    PROC StoreSlot_P04(num slot, num subType, num toolSel, num lenMM,
                       robtarget arcStart, robtarget arcEnd, robtarget approach, robtarget retract, robtarget trans)
        IF slot = 1 THEN
            P04W01_SubType := subType;
            P04W01_ToolSel := toolSel;
            P04W01_LenMM := lenMM;
            P04W01_ArcStart := arcStart;
            P04W01_ArcEnd := arcEnd;
            P04W01_Approach := approach;
            P04W01_Retract := retract;
            P04W01_Trans := trans;
            P04W01_Used := TRUE;
        ELSEIF slot = 2 THEN
            P04W02_SubType := subType;
            P04W02_ToolSel := toolSel;
            P04W02_LenMM := lenMM;
            P04W02_ArcStart := arcStart;
            P04W02_ArcEnd := arcEnd;
            P04W02_Approach := approach;
            P04W02_Retract := retract;
            P04W02_Trans := trans;
            P04W02_Used := TRUE;
        ELSEIF slot = 3 THEN
            P04W03_SubType := subType;
            P04W03_ToolSel := toolSel;
            P04W03_LenMM := lenMM;
            P04W03_ArcStart := arcStart;
            P04W03_ArcEnd := arcEnd;
            P04W03_Approach := approach;
            P04W03_Retract := retract;
            P04W03_Trans := trans;
            P04W03_Used := TRUE;
        ELSEIF slot = 4 THEN
            P04W04_SubType := subType;
            P04W04_ToolSel := toolSel;
            P04W04_LenMM := lenMM;
            P04W04_ArcStart := arcStart;
            P04W04_ArcEnd := arcEnd;
            P04W04_Approach := approach;
            P04W04_Retract := retract;
            P04W04_Trans := trans;
            P04W04_Used := TRUE;
        ELSEIF slot = 5 THEN
            P04W05_SubType := subType;
            P04W05_ToolSel := toolSel;
            P04W05_LenMM := lenMM;
            P04W05_ArcStart := arcStart;
            P04W05_ArcEnd := arcEnd;
            P04W05_Approach := approach;
            P04W05_Retract := retract;
            P04W05_Trans := trans;
            P04W05_Used := TRUE;
        ELSEIF slot = 6 THEN
            P04W06_SubType := subType;
            P04W06_ToolSel := toolSel;
            P04W06_LenMM := lenMM;
            P04W06_ArcStart := arcStart;
            P04W06_ArcEnd := arcEnd;
            P04W06_Approach := approach;
            P04W06_Retract := retract;
            P04W06_Trans := trans;
            P04W06_Used := TRUE;
        ELSEIF slot = 7 THEN
            P04W07_SubType := subType;
            P04W07_ToolSel := toolSel;
            P04W07_LenMM := lenMM;
            P04W07_ArcStart := arcStart;
            P04W07_ArcEnd := arcEnd;
            P04W07_Approach := approach;
            P04W07_Retract := retract;
            P04W07_Trans := trans;
            P04W07_Used := TRUE;
        ELSEIF slot = 8 THEN
            P04W08_SubType := subType;
            P04W08_ToolSel := toolSel;
            P04W08_LenMM := lenMM;
            P04W08_ArcStart := arcStart;
            P04W08_ArcEnd := arcEnd;
            P04W08_Approach := approach;
            P04W08_Retract := retract;
            P04W08_Trans := trans;
            P04W08_Used := TRUE;
        ELSEIF slot = 9 THEN
            P04W09_SubType := subType;
            P04W09_ToolSel := toolSel;
            P04W09_LenMM := lenMM;
            P04W09_ArcStart := arcStart;
            P04W09_ArcEnd := arcEnd;
            P04W09_Approach := approach;
            P04W09_Retract := retract;
            P04W09_Trans := trans;
            P04W09_Used := TRUE;
        ELSEIF slot = 10 THEN
            P04W10_SubType := subType;
            P04W10_ToolSel := toolSel;
            P04W10_LenMM := lenMM;
            P04W10_ArcStart := arcStart;
            P04W10_ArcEnd := arcEnd;
            P04W10_Approach := approach;
            P04W10_Retract := retract;
            P04W10_Trans := trans;
            P04W10_Used := TRUE;
        ELSEIF slot = 11 THEN
            P04W11_SubType := subType;
            P04W11_ToolSel := toolSel;
            P04W11_LenMM := lenMM;
            P04W11_ArcStart := arcStart;
            P04W11_ArcEnd := arcEnd;
            P04W11_Approach := approach;
            P04W11_Retract := retract;
            P04W11_Trans := trans;
            P04W11_Used := TRUE;
        ELSEIF slot = 12 THEN
            P04W12_SubType := subType;
            P04W12_ToolSel := toolSel;
            P04W12_LenMM := lenMM;
            P04W12_ArcStart := arcStart;
            P04W12_ArcEnd := arcEnd;
            P04W12_Approach := approach;
            P04W12_Retract := retract;
            P04W12_Trans := trans;
            P04W12_Used := TRUE;
        ELSEIF slot = 13 THEN
            P04W13_SubType := subType;
            P04W13_ToolSel := toolSel;
            P04W13_LenMM := lenMM;
            P04W13_ArcStart := arcStart;
            P04W13_ArcEnd := arcEnd;
            P04W13_Approach := approach;
            P04W13_Retract := retract;
            P04W13_Trans := trans;
            P04W13_Used := TRUE;
        ELSEIF slot = 14 THEN
            P04W14_SubType := subType;
            P04W14_ToolSel := toolSel;
            P04W14_LenMM := lenMM;
            P04W14_ArcStart := arcStart;
            P04W14_ArcEnd := arcEnd;
            P04W14_Approach := approach;
            P04W14_Retract := retract;
            P04W14_Trans := trans;
            P04W14_Used := TRUE;
        ELSEIF slot = 15 THEN
            P04W15_SubType := subType;
            P04W15_ToolSel := toolSel;
            P04W15_LenMM := lenMM;
            P04W15_ArcStart := arcStart;
            P04W15_ArcEnd := arcEnd;
            P04W15_Approach := approach;
            P04W15_Retract := retract;
            P04W15_Trans := trans;
            P04W15_Used := TRUE;
        ELSEIF slot = 16 THEN
            P04W16_SubType := subType;
            P04W16_ToolSel := toolSel;
            P04W16_LenMM := lenMM;
            P04W16_ArcStart := arcStart;
            P04W16_ArcEnd := arcEnd;
            P04W16_Approach := approach;
            P04W16_Retract := retract;
            P04W16_Trans := trans;
            P04W16_Used := TRUE;
        ELSEIF slot = 17 THEN
            P04W17_SubType := subType;
            P04W17_ToolSel := toolSel;
            P04W17_LenMM := lenMM;
            P04W17_ArcStart := arcStart;
            P04W17_ArcEnd := arcEnd;
            P04W17_Approach := approach;
            P04W17_Retract := retract;
            P04W17_Trans := trans;
            P04W17_Used := TRUE;
        ELSEIF slot = 18 THEN
            P04W18_SubType := subType;
            P04W18_ToolSel := toolSel;
            P04W18_LenMM := lenMM;
            P04W18_ArcStart := arcStart;
            P04W18_ArcEnd := arcEnd;
            P04W18_Approach := approach;
            P04W18_Retract := retract;
            P04W18_Trans := trans;
            P04W18_Used := TRUE;
        ELSEIF slot = 19 THEN
            P04W19_SubType := subType;
            P04W19_ToolSel := toolSel;
            P04W19_LenMM := lenMM;
            P04W19_ArcStart := arcStart;
            P04W19_ArcEnd := arcEnd;
            P04W19_Approach := approach;
            P04W19_Retract := retract;
            P04W19_Trans := trans;
            P04W19_Used := TRUE;
        ELSEIF slot = 20 THEN
            P04W20_SubType := subType;
            P04W20_ToolSel := toolSel;
            P04W20_LenMM := lenMM;
            P04W20_ArcStart := arcStart;
            P04W20_ArcEnd := arcEnd;
            P04W20_Approach := approach;
            P04W20_Retract := retract;
            P04W20_Trans := trans;
            P04W20_Used := TRUE;
        ELSEIF slot = 21 THEN
            P04W21_SubType := subType;
            P04W21_ToolSel := toolSel;
            P04W21_LenMM := lenMM;
            P04W21_ArcStart := arcStart;
            P04W21_ArcEnd := arcEnd;
            P04W21_Approach := approach;
            P04W21_Retract := retract;
            P04W21_Trans := trans;
            P04W21_Used := TRUE;
        ELSEIF slot = 22 THEN
            P04W22_SubType := subType;
            P04W22_ToolSel := toolSel;
            P04W22_LenMM := lenMM;
            P04W22_ArcStart := arcStart;
            P04W22_ArcEnd := arcEnd;
            P04W22_Approach := approach;
            P04W22_Retract := retract;
            P04W22_Trans := trans;
            P04W22_Used := TRUE;
        ELSEIF slot = 23 THEN
            P04W23_SubType := subType;
            P04W23_ToolSel := toolSel;
            P04W23_LenMM := lenMM;
            P04W23_ArcStart := arcStart;
            P04W23_ArcEnd := arcEnd;
            P04W23_Approach := approach;
            P04W23_Retract := retract;
            P04W23_Trans := trans;
            P04W23_Used := TRUE;
        ELSEIF slot = 24 THEN
            P04W24_SubType := subType;
            P04W24_ToolSel := toolSel;
            P04W24_LenMM := lenMM;
            P04W24_ArcStart := arcStart;
            P04W24_ArcEnd := arcEnd;
            P04W24_Approach := approach;
            P04W24_Retract := retract;
            P04W24_Trans := trans;
            P04W24_Used := TRUE;
        ELSEIF slot = 25 THEN
            P04W25_SubType := subType;
            P04W25_ToolSel := toolSel;
            P04W25_LenMM := lenMM;
            P04W25_ArcStart := arcStart;
            P04W25_ArcEnd := arcEnd;
            P04W25_Approach := approach;
            P04W25_Retract := retract;
            P04W25_Trans := trans;
            P04W25_Used := TRUE;
        ELSEIF slot = 26 THEN
            P04W26_SubType := subType;
            P04W26_ToolSel := toolSel;
            P04W26_LenMM := lenMM;
            P04W26_ArcStart := arcStart;
            P04W26_ArcEnd := arcEnd;
            P04W26_Approach := approach;
            P04W26_Retract := retract;
            P04W26_Trans := trans;
            P04W26_Used := TRUE;
        ELSEIF slot = 27 THEN
            P04W27_SubType := subType;
            P04W27_ToolSel := toolSel;
            P04W27_LenMM := lenMM;
            P04W27_ArcStart := arcStart;
            P04W27_ArcEnd := arcEnd;
            P04W27_Approach := approach;
            P04W27_Retract := retract;
            P04W27_Trans := trans;
            P04W27_Used := TRUE;
        ELSEIF slot = 28 THEN
            P04W28_SubType := subType;
            P04W28_ToolSel := toolSel;
            P04W28_LenMM := lenMM;
            P04W28_ArcStart := arcStart;
            P04W28_ArcEnd := arcEnd;
            P04W28_Approach := approach;
            P04W28_Retract := retract;
            P04W28_Trans := trans;
            P04W28_Used := TRUE;
        ELSEIF slot = 29 THEN
            P04W29_SubType := subType;
            P04W29_ToolSel := toolSel;
            P04W29_LenMM := lenMM;
            P04W29_ArcStart := arcStart;
            P04W29_ArcEnd := arcEnd;
            P04W29_Approach := approach;
            P04W29_Retract := retract;
            P04W29_Trans := trans;
            P04W29_Used := TRUE;
        ELSEIF slot = 30 THEN
            P04W30_SubType := subType;
            P04W30_ToolSel := toolSel;
            P04W30_LenMM := lenMM;
            P04W30_ArcStart := arcStart;
            P04W30_ArcEnd := arcEnd;
            P04W30_Approach := approach;
            P04W30_Retract := retract;
            P04W30_Trans := trans;
            P04W30_Used := TRUE;
        ELSE
            TPWrite "Invalid weld slot.";
        ENDIF
    ENDPROC

    PROC LoadSlot_P04(num slot, VAR bool used, VAR num subType, VAR num toolSel, VAR num lenMM,
                       VAR robtarget arcStart, VAR robtarget arcEnd, VAR robtarget approach, VAR robtarget retract, VAR robtarget trans)
        IF slot = 1 THEN
            used := P04W01_Used;
            subType := P04W01_SubType;
            toolSel := P04W01_ToolSel;
            lenMM := P04W01_LenMM;
            arcStart := P04W01_ArcStart;
            arcEnd := P04W01_ArcEnd;
            approach := P04W01_Approach;
            retract := P04W01_Retract;
            trans := P04W01_Trans;
        ELSEIF slot = 2 THEN
            used := P04W02_Used;
            subType := P04W02_SubType;
            toolSel := P04W02_ToolSel;
            lenMM := P04W02_LenMM;
            arcStart := P04W02_ArcStart;
            arcEnd := P04W02_ArcEnd;
            approach := P04W02_Approach;
            retract := P04W02_Retract;
            trans := P04W02_Trans;
        ELSEIF slot = 3 THEN
            used := P04W03_Used;
            subType := P04W03_SubType;
            toolSel := P04W03_ToolSel;
            lenMM := P04W03_LenMM;
            arcStart := P04W03_ArcStart;
            arcEnd := P04W03_ArcEnd;
            approach := P04W03_Approach;
            retract := P04W03_Retract;
            trans := P04W03_Trans;
        ELSEIF slot = 4 THEN
            used := P04W04_Used;
            subType := P04W04_SubType;
            toolSel := P04W04_ToolSel;
            lenMM := P04W04_LenMM;
            arcStart := P04W04_ArcStart;
            arcEnd := P04W04_ArcEnd;
            approach := P04W04_Approach;
            retract := P04W04_Retract;
            trans := P04W04_Trans;
        ELSEIF slot = 5 THEN
            used := P04W05_Used;
            subType := P04W05_SubType;
            toolSel := P04W05_ToolSel;
            lenMM := P04W05_LenMM;
            arcStart := P04W05_ArcStart;
            arcEnd := P04W05_ArcEnd;
            approach := P04W05_Approach;
            retract := P04W05_Retract;
            trans := P04W05_Trans;
        ELSEIF slot = 6 THEN
            used := P04W06_Used;
            subType := P04W06_SubType;
            toolSel := P04W06_ToolSel;
            lenMM := P04W06_LenMM;
            arcStart := P04W06_ArcStart;
            arcEnd := P04W06_ArcEnd;
            approach := P04W06_Approach;
            retract := P04W06_Retract;
            trans := P04W06_Trans;
        ELSEIF slot = 7 THEN
            used := P04W07_Used;
            subType := P04W07_SubType;
            toolSel := P04W07_ToolSel;
            lenMM := P04W07_LenMM;
            arcStart := P04W07_ArcStart;
            arcEnd := P04W07_ArcEnd;
            approach := P04W07_Approach;
            retract := P04W07_Retract;
            trans := P04W07_Trans;
        ELSEIF slot = 8 THEN
            used := P04W08_Used;
            subType := P04W08_SubType;
            toolSel := P04W08_ToolSel;
            lenMM := P04W08_LenMM;
            arcStart := P04W08_ArcStart;
            arcEnd := P04W08_ArcEnd;
            approach := P04W08_Approach;
            retract := P04W08_Retract;
            trans := P04W08_Trans;
        ELSEIF slot = 9 THEN
            used := P04W09_Used;
            subType := P04W09_SubType;
            toolSel := P04W09_ToolSel;
            lenMM := P04W09_LenMM;
            arcStart := P04W09_ArcStart;
            arcEnd := P04W09_ArcEnd;
            approach := P04W09_Approach;
            retract := P04W09_Retract;
            trans := P04W09_Trans;
        ELSEIF slot = 10 THEN
            used := P04W10_Used;
            subType := P04W10_SubType;
            toolSel := P04W10_ToolSel;
            lenMM := P04W10_LenMM;
            arcStart := P04W10_ArcStart;
            arcEnd := P04W10_ArcEnd;
            approach := P04W10_Approach;
            retract := P04W10_Retract;
            trans := P04W10_Trans;
        ELSEIF slot = 11 THEN
            used := P04W11_Used;
            subType := P04W11_SubType;
            toolSel := P04W11_ToolSel;
            lenMM := P04W11_LenMM;
            arcStart := P04W11_ArcStart;
            arcEnd := P04W11_ArcEnd;
            approach := P04W11_Approach;
            retract := P04W11_Retract;
            trans := P04W11_Trans;
        ELSEIF slot = 12 THEN
            used := P04W12_Used;
            subType := P04W12_SubType;
            toolSel := P04W12_ToolSel;
            lenMM := P04W12_LenMM;
            arcStart := P04W12_ArcStart;
            arcEnd := P04W12_ArcEnd;
            approach := P04W12_Approach;
            retract := P04W12_Retract;
            trans := P04W12_Trans;
        ELSEIF slot = 13 THEN
            used := P04W13_Used;
            subType := P04W13_SubType;
            toolSel := P04W13_ToolSel;
            lenMM := P04W13_LenMM;
            arcStart := P04W13_ArcStart;
            arcEnd := P04W13_ArcEnd;
            approach := P04W13_Approach;
            retract := P04W13_Retract;
            trans := P04W13_Trans;
        ELSEIF slot = 14 THEN
            used := P04W14_Used;
            subType := P04W14_SubType;
            toolSel := P04W14_ToolSel;
            lenMM := P04W14_LenMM;
            arcStart := P04W14_ArcStart;
            arcEnd := P04W14_ArcEnd;
            approach := P04W14_Approach;
            retract := P04W14_Retract;
            trans := P04W14_Trans;
        ELSEIF slot = 15 THEN
            used := P04W15_Used;
            subType := P04W15_SubType;
            toolSel := P04W15_ToolSel;
            lenMM := P04W15_LenMM;
            arcStart := P04W15_ArcStart;
            arcEnd := P04W15_ArcEnd;
            approach := P04W15_Approach;
            retract := P04W15_Retract;
            trans := P04W15_Trans;
        ELSEIF slot = 16 THEN
            used := P04W16_Used;
            subType := P04W16_SubType;
            toolSel := P04W16_ToolSel;
            lenMM := P04W16_LenMM;
            arcStart := P04W16_ArcStart;
            arcEnd := P04W16_ArcEnd;
            approach := P04W16_Approach;
            retract := P04W16_Retract;
            trans := P04W16_Trans;
        ELSEIF slot = 17 THEN
            used := P04W17_Used;
            subType := P04W17_SubType;
            toolSel := P04W17_ToolSel;
            lenMM := P04W17_LenMM;
            arcStart := P04W17_ArcStart;
            arcEnd := P04W17_ArcEnd;
            approach := P04W17_Approach;
            retract := P04W17_Retract;
            trans := P04W17_Trans;
        ELSEIF slot = 18 THEN
            used := P04W18_Used;
            subType := P04W18_SubType;
            toolSel := P04W18_ToolSel;
            lenMM := P04W18_LenMM;
            arcStart := P04W18_ArcStart;
            arcEnd := P04W18_ArcEnd;
            approach := P04W18_Approach;
            retract := P04W18_Retract;
            trans := P04W18_Trans;
        ELSEIF slot = 19 THEN
            used := P04W19_Used;
            subType := P04W19_SubType;
            toolSel := P04W19_ToolSel;
            lenMM := P04W19_LenMM;
            arcStart := P04W19_ArcStart;
            arcEnd := P04W19_ArcEnd;
            approach := P04W19_Approach;
            retract := P04W19_Retract;
            trans := P04W19_Trans;
        ELSEIF slot = 20 THEN
            used := P04W20_Used;
            subType := P04W20_SubType;
            toolSel := P04W20_ToolSel;
            lenMM := P04W20_LenMM;
            arcStart := P04W20_ArcStart;
            arcEnd := P04W20_ArcEnd;
            approach := P04W20_Approach;
            retract := P04W20_Retract;
            trans := P04W20_Trans;
        ELSEIF slot = 21 THEN
            used := P04W21_Used;
            subType := P04W21_SubType;
            toolSel := P04W21_ToolSel;
            lenMM := P04W21_LenMM;
            arcStart := P04W21_ArcStart;
            arcEnd := P04W21_ArcEnd;
            approach := P04W21_Approach;
            retract := P04W21_Retract;
            trans := P04W21_Trans;
        ELSEIF slot = 22 THEN
            used := P04W22_Used;
            subType := P04W22_SubType;
            toolSel := P04W22_ToolSel;
            lenMM := P04W22_LenMM;
            arcStart := P04W22_ArcStart;
            arcEnd := P04W22_ArcEnd;
            approach := P04W22_Approach;
            retract := P04W22_Retract;
            trans := P04W22_Trans;
        ELSEIF slot = 23 THEN
            used := P04W23_Used;
            subType := P04W23_SubType;
            toolSel := P04W23_ToolSel;
            lenMM := P04W23_LenMM;
            arcStart := P04W23_ArcStart;
            arcEnd := P04W23_ArcEnd;
            approach := P04W23_Approach;
            retract := P04W23_Retract;
            trans := P04W23_Trans;
        ELSEIF slot = 24 THEN
            used := P04W24_Used;
            subType := P04W24_SubType;
            toolSel := P04W24_ToolSel;
            lenMM := P04W24_LenMM;
            arcStart := P04W24_ArcStart;
            arcEnd := P04W24_ArcEnd;
            approach := P04W24_Approach;
            retract := P04W24_Retract;
            trans := P04W24_Trans;
        ELSEIF slot = 25 THEN
            used := P04W25_Used;
            subType := P04W25_SubType;
            toolSel := P04W25_ToolSel;
            lenMM := P04W25_LenMM;
            arcStart := P04W25_ArcStart;
            arcEnd := P04W25_ArcEnd;
            approach := P04W25_Approach;
            retract := P04W25_Retract;
            trans := P04W25_Trans;
        ELSEIF slot = 26 THEN
            used := P04W26_Used;
            subType := P04W26_SubType;
            toolSel := P04W26_ToolSel;
            lenMM := P04W26_LenMM;
            arcStart := P04W26_ArcStart;
            arcEnd := P04W26_ArcEnd;
            approach := P04W26_Approach;
            retract := P04W26_Retract;
            trans := P04W26_Trans;
        ELSEIF slot = 27 THEN
            used := P04W27_Used;
            subType := P04W27_SubType;
            toolSel := P04W27_ToolSel;
            lenMM := P04W27_LenMM;
            arcStart := P04W27_ArcStart;
            arcEnd := P04W27_ArcEnd;
            approach := P04W27_Approach;
            retract := P04W27_Retract;
            trans := P04W27_Trans;
        ELSEIF slot = 28 THEN
            used := P04W28_Used;
            subType := P04W28_SubType;
            toolSel := P04W28_ToolSel;
            lenMM := P04W28_LenMM;
            arcStart := P04W28_ArcStart;
            arcEnd := P04W28_ArcEnd;
            approach := P04W28_Approach;
            retract := P04W28_Retract;
            trans := P04W28_Trans;
        ELSEIF slot = 29 THEN
            used := P04W29_Used;
            subType := P04W29_SubType;
            toolSel := P04W29_ToolSel;
            lenMM := P04W29_LenMM;
            arcStart := P04W29_ArcStart;
            arcEnd := P04W29_ArcEnd;
            approach := P04W29_Approach;
            retract := P04W29_Retract;
            trans := P04W29_Trans;
        ELSEIF slot = 30 THEN
            used := P04W30_Used;
            subType := P04W30_SubType;
            toolSel := P04W30_ToolSel;
            lenMM := P04W30_LenMM;
            arcStart := P04W30_ArcStart;
            arcEnd := P04W30_ArcEnd;
            approach := P04W30_Approach;
            retract := P04W30_Retract;
            trans := P04W30_Trans;
        ELSE
            used := FALSE;
        ENDIF
    ENDPROC

    PROC ClearSlot_P04(num slot)
        IF slot = 1 THEN
            P04W01_Used := FALSE;
            P04W01_SubType := 0;
            P04W01_ToolSel := 0;
            P04W01_LenMM := 0;
            P04W01_ArcStart := [[0,0,0],[1,0,0,0],[0,0,0,0],[9E9,9E9,9E9,9E9,9E9,9E9]];
            P04W01_ArcEnd := [[0,0,0],[1,0,0,0],[0,0,0,0],[9E9,9E9,9E9,9E9,9E9,9E9]];
            P04W01_Approach := [[0,0,0],[1,0,0,0],[0,0,0,0],[9E9,9E9,9E9,9E9,9E9,9E9]];
            P04W01_Retract := [[0,0,0],[1,0,0,0],[0,0,0,0],[9E9,9E9,9E9,9E9,9E9,9E9]];
            P04W01_Trans := [[0,0,0],[1,0,0,0],[0,0,0,0],[9E9,9E9,9E9,9E9,9E9,9E9]];
        ELSEIF slot = 2 THEN
            P04W02_Used := FALSE;
            P04W02_SubType := 0;
            P04W02_ToolSel := 0;
            P04W02_LenMM := 0;
            P04W02_ArcStart := [[0,0,0],[1,0,0,0],[0,0,0,0],[9E9,9E9,9E9,9E9,9E9,9E9]];
            P04W02_ArcEnd := [[0,0,0],[1,0,0,0],[0,0,0,0],[9E9,9E9,9E9,9E9,9E9,9E9]];
            P04W02_Approach := [[0,0,0],[1,0,0,0],[0,0,0,0],[9E9,9E9,9E9,9E9,9E9,9E9]];
            P04W02_Retract := [[0,0,0],[1,0,0,0],[0,0,0,0],[9E9,9E9,9E9,9E9,9E9,9E9]];
            P04W02_Trans := [[0,0,0],[1,0,0,0],[0,0,0,0],[9E9,9E9,9E9,9E9,9E9,9E9]];
        ELSEIF slot = 3 THEN
            P04W03_Used := FALSE;
            P04W03_SubType := 0;
            P04W03_ToolSel := 0;
            P04W03_LenMM := 0;
            P04W03_ArcStart := [[0,0,0],[1,0,0,0],[0,0,0,0],[9E9,9E9,9E9,9E9,9E9,9E9]];
            P04W03_ArcEnd := [[0,0,0],[1,0,0,0],[0,0,0,0],[9E9,9E9,9E9,9E9,9E9,9E9]];
            P04W03_Approach := [[0,0,0],[1,0,0,0],[0,0,0,0],[9E9,9E9,9E9,9E9,9E9,9E9]];
            P04W03_Retract := [[0,0,0],[1,0,0,0],[0,0,0,0],[9E9,9E9,9E9,9E9,9E9,9E9]];
            P04W03_Trans := [[0,0,0],[1,0,0,0],[0,0,0,0],[9E9,9E9,9E9,9E9,9E9,9E9]];
        ELSEIF slot = 4 THEN
            P04W04_Used := FALSE;
            P04W04_SubType := 0;
            P04W04_ToolSel := 0;
            P04W04_LenMM := 0;
            P04W04_ArcStart := [[0,0,0],[1,0,0,0],[0,0,0,0],[9E9,9E9,9E9,9E9,9E9,9E9]];
            P04W04_ArcEnd := [[0,0,0],[1,0,0,0],[0,0,0,0],[9E9,9E9,9E9,9E9,9E9,9E9]];
            P04W04_Approach := [[0,0,0],[1,0,0,0],[0,0,0,0],[9E9,9E9,9E9,9E9,9E9,9E9]];
            P04W04_Retract := [[0,0,0],[1,0,0,0],[0,0,0,0],[9E9,9E9,9E9,9E9,9E9,9E9]];
            P04W04_Trans := [[0,0,0],[1,0,0,0],[0,0,0,0],[9E9,9E9,9E9,9E9,9E9,9E9]];
        ELSEIF slot = 5 THEN
            P04W05_Used := FALSE;
            P04W05_SubType := 0;
            P04W05_ToolSel := 0;
            P04W05_LenMM := 0;
            P04W05_ArcStart := [[0,0,0],[1,0,0,0],[0,0,0,0],[9E9,9E9,9E9,9E9,9E9,9E9]];
            P04W05_ArcEnd := [[0,0,0],[1,0,0,0],[0,0,0,0],[9E9,9E9,9E9,9E9,9E9,9E9]];
            P04W05_Approach := [[0,0,0],[1,0,0,0],[0,0,0,0],[9E9,9E9,9E9,9E9,9E9,9E9]];
            P04W05_Retract := [[0,0,0],[1,0,0,0],[0,0,0,0],[9E9,9E9,9E9,9E9,9E9,9E9]];
            P04W05_Trans := [[0,0,0],[1,0,0,0],[0,0,0,0],[9E9,9E9,9E9,9E9,9E9,9E9]];
        ELSEIF slot = 6 THEN
            P04W06_Used := FALSE;
            P04W06_SubType := 0;
            P04W06_ToolSel := 0;
            P04W06_LenMM := 0;
            P04W06_ArcStart := [[0,0,0],[1,0,0,0],[0,0,0,0],[9E9,9E9,9E9,9E9,9E9,9E9]];
            P04W06_ArcEnd := [[0,0,0],[1,0,0,0],[0,0,0,0],[9E9,9E9,9E9,9E9,9E9,9E9]];
            P04W06_Approach := [[0,0,0],[1,0,0,0],[0,0,0,0],[9E9,9E9,9E9,9E9,9E9,9E9]];
            P04W06_Retract := [[0,0,0],[1,0,0,0],[0,0,0,0],[9E9,9E9,9E9,9E9,9E9,9E9]];
            P04W06_Trans := [[0,0,0],[1,0,0,0],[0,0,0,0],[9E9,9E9,9E9,9E9,9E9,9E9]];
        ELSEIF slot = 7 THEN
            P04W07_Used := FALSE;
            P04W07_SubType := 0;
            P04W07_ToolSel := 0;
            P04W07_LenMM := 0;
            P04W07_ArcStart := [[0,0,0],[1,0,0,0],[0,0,0,0],[9E9,9E9,9E9,9E9,9E9,9E9]];
            P04W07_ArcEnd := [[0,0,0],[1,0,0,0],[0,0,0,0],[9E9,9E9,9E9,9E9,9E9,9E9]];
            P04W07_Approach := [[0,0,0],[1,0,0,0],[0,0,0,0],[9E9,9E9,9E9,9E9,9E9,9E9]];
            P04W07_Retract := [[0,0,0],[1,0,0,0],[0,0,0,0],[9E9,9E9,9E9,9E9,9E9,9E9]];
            P04W07_Trans := [[0,0,0],[1,0,0,0],[0,0,0,0],[9E9,9E9,9E9,9E9,9E9,9E9]];
        ELSEIF slot = 8 THEN
            P04W08_Used := FALSE;
            P04W08_SubType := 0;
            P04W08_ToolSel := 0;
            P04W08_LenMM := 0;
            P04W08_ArcStart := [[0,0,0],[1,0,0,0],[0,0,0,0],[9E9,9E9,9E9,9E9,9E9,9E9]];
            P04W08_ArcEnd := [[0,0,0],[1,0,0,0],[0,0,0,0],[9E9,9E9,9E9,9E9,9E9,9E9]];
            P04W08_Approach := [[0,0,0],[1,0,0,0],[0,0,0,0],[9E9,9E9,9E9,9E9,9E9,9E9]];
            P04W08_Retract := [[0,0,0],[1,0,0,0],[0,0,0,0],[9E9,9E9,9E9,9E9,9E9,9E9]];
            P04W08_Trans := [[0,0,0],[1,0,0,0],[0,0,0,0],[9E9,9E9,9E9,9E9,9E9,9E9]];
        ELSEIF slot = 9 THEN
            P04W09_Used := FALSE;
            P04W09_SubType := 0;
            P04W09_ToolSel := 0;
            P04W09_LenMM := 0;
            P04W09_ArcStart := [[0,0,0],[1,0,0,0],[0,0,0,0],[9E9,9E9,9E9,9E9,9E9,9E9]];
            P04W09_ArcEnd := [[0,0,0],[1,0,0,0],[0,0,0,0],[9E9,9E9,9E9,9E9,9E9,9E9]];
            P04W09_Approach := [[0,0,0],[1,0,0,0],[0,0,0,0],[9E9,9E9,9E9,9E9,9E9,9E9]];
            P04W09_Retract := [[0,0,0],[1,0,0,0],[0,0,0,0],[9E9,9E9,9E9,9E9,9E9,9E9]];
            P04W09_Trans := [[0,0,0],[1,0,0,0],[0,0,0,0],[9E9,9E9,9E9,9E9,9E9,9E9]];
        ELSEIF slot = 10 THEN
            P04W10_Used := FALSE;
            P04W10_SubType := 0;
            P04W10_ToolSel := 0;
            P04W10_LenMM := 0;
            P04W10_ArcStart := [[0,0,0],[1,0,0,0],[0,0,0,0],[9E9,9E9,9E9,9E9,9E9,9E9]];
            P04W10_ArcEnd := [[0,0,0],[1,0,0,0],[0,0,0,0],[9E9,9E9,9E9,9E9,9E9,9E9]];
            P04W10_Approach := [[0,0,0],[1,0,0,0],[0,0,0,0],[9E9,9E9,9E9,9E9,9E9,9E9]];
            P04W10_Retract := [[0,0,0],[1,0,0,0],[0,0,0,0],[9E9,9E9,9E9,9E9,9E9,9E9]];
            P04W10_Trans := [[0,0,0],[1,0,0,0],[0,0,0,0],[9E9,9E9,9E9,9E9,9E9,9E9]];
        ELSEIF slot = 11 THEN
            P04W11_Used := FALSE;
            P04W11_SubType := 0;
            P04W11_ToolSel := 0;
            P04W11_LenMM := 0;
            P04W11_ArcStart := [[0,0,0],[1,0,0,0],[0,0,0,0],[9E9,9E9,9E9,9E9,9E9,9E9]];
            P04W11_ArcEnd := [[0,0,0],[1,0,0,0],[0,0,0,0],[9E9,9E9,9E9,9E9,9E9,9E9]];
            P04W11_Approach := [[0,0,0],[1,0,0,0],[0,0,0,0],[9E9,9E9,9E9,9E9,9E9,9E9]];
            P04W11_Retract := [[0,0,0],[1,0,0,0],[0,0,0,0],[9E9,9E9,9E9,9E9,9E9,9E9]];
            P04W11_Trans := [[0,0,0],[1,0,0,0],[0,0,0,0],[9E9,9E9,9E9,9E9,9E9,9E9]];
        ELSEIF slot = 12 THEN
            P04W12_Used := FALSE;
            P04W12_SubType := 0;
            P04W12_ToolSel := 0;
            P04W12_LenMM := 0;
            P04W12_ArcStart := [[0,0,0],[1,0,0,0],[0,0,0,0],[9E9,9E9,9E9,9E9,9E9,9E9]];
            P04W12_ArcEnd := [[0,0,0],[1,0,0,0],[0,0,0,0],[9E9,9E9,9E9,9E9,9E9,9E9]];
            P04W12_Approach := [[0,0,0],[1,0,0,0],[0,0,0,0],[9E9,9E9,9E9,9E9,9E9,9E9]];
            P04W12_Retract := [[0,0,0],[1,0,0,0],[0,0,0,0],[9E9,9E9,9E9,9E9,9E9,9E9]];
            P04W12_Trans := [[0,0,0],[1,0,0,0],[0,0,0,0],[9E9,9E9,9E9,9E9,9E9,9E9]];
        ELSEIF slot = 13 THEN
            P04W13_Used := FALSE;
            P04W13_SubType := 0;
            P04W13_ToolSel := 0;
            P04W13_LenMM := 0;
            P04W13_ArcStart := [[0,0,0],[1,0,0,0],[0,0,0,0],[9E9,9E9,9E9,9E9,9E9,9E9]];
            P04W13_ArcEnd := [[0,0,0],[1,0,0,0],[0,0,0,0],[9E9,9E9,9E9,9E9,9E9,9E9]];
            P04W13_Approach := [[0,0,0],[1,0,0,0],[0,0,0,0],[9E9,9E9,9E9,9E9,9E9,9E9]];
            P04W13_Retract := [[0,0,0],[1,0,0,0],[0,0,0,0],[9E9,9E9,9E9,9E9,9E9,9E9]];
            P04W13_Trans := [[0,0,0],[1,0,0,0],[0,0,0,0],[9E9,9E9,9E9,9E9,9E9,9E9]];
        ELSEIF slot = 14 THEN
            P04W14_Used := FALSE;
            P04W14_SubType := 0;
            P04W14_ToolSel := 0;
            P04W14_LenMM := 0;
            P04W14_ArcStart := [[0,0,0],[1,0,0,0],[0,0,0,0],[9E9,9E9,9E9,9E9,9E9,9E9]];
            P04W14_ArcEnd := [[0,0,0],[1,0,0,0],[0,0,0,0],[9E9,9E9,9E9,9E9,9E9,9E9]];
            P04W14_Approach := [[0,0,0],[1,0,0,0],[0,0,0,0],[9E9,9E9,9E9,9E9,9E9,9E9]];
            P04W14_Retract := [[0,0,0],[1,0,0,0],[0,0,0,0],[9E9,9E9,9E9,9E9,9E9,9E9]];
            P04W14_Trans := [[0,0,0],[1,0,0,0],[0,0,0,0],[9E9,9E9,9E9,9E9,9E9,9E9]];
        ELSEIF slot = 15 THEN
            P04W15_Used := FALSE;
            P04W15_SubType := 0;
            P04W15_ToolSel := 0;
            P04W15_LenMM := 0;
            P04W15_ArcStart := [[0,0,0],[1,0,0,0],[0,0,0,0],[9E9,9E9,9E9,9E9,9E9,9E9]];
            P04W15_ArcEnd := [[0,0,0],[1,0,0,0],[0,0,0,0],[9E9,9E9,9E9,9E9,9E9,9E9]];
            P04W15_Approach := [[0,0,0],[1,0,0,0],[0,0,0,0],[9E9,9E9,9E9,9E9,9E9,9E9]];
            P04W15_Retract := [[0,0,0],[1,0,0,0],[0,0,0,0],[9E9,9E9,9E9,9E9,9E9,9E9]];
            P04W15_Trans := [[0,0,0],[1,0,0,0],[0,0,0,0],[9E9,9E9,9E9,9E9,9E9,9E9]];
        ELSEIF slot = 16 THEN
            P04W16_Used := FALSE;
            P04W16_SubType := 0;
            P04W16_ToolSel := 0;
            P04W16_LenMM := 0;
            P04W16_ArcStart := [[0,0,0],[1,0,0,0],[0,0,0,0],[9E9,9E9,9E9,9E9,9E9,9E9]];
            P04W16_ArcEnd := [[0,0,0],[1,0,0,0],[0,0,0,0],[9E9,9E9,9E9,9E9,9E9,9E9]];
            P04W16_Approach := [[0,0,0],[1,0,0,0],[0,0,0,0],[9E9,9E9,9E9,9E9,9E9,9E9]];
            P04W16_Retract := [[0,0,0],[1,0,0,0],[0,0,0,0],[9E9,9E9,9E9,9E9,9E9,9E9]];
            P04W16_Trans := [[0,0,0],[1,0,0,0],[0,0,0,0],[9E9,9E9,9E9,9E9,9E9,9E9]];
        ELSEIF slot = 17 THEN
            P04W17_Used := FALSE;
            P04W17_SubType := 0;
            P04W17_ToolSel := 0;
            P04W17_LenMM := 0;
            P04W17_ArcStart := [[0,0,0],[1,0,0,0],[0,0,0,0],[9E9,9E9,9E9,9E9,9E9,9E9]];
            P04W17_ArcEnd := [[0,0,0],[1,0,0,0],[0,0,0,0],[9E9,9E9,9E9,9E9,9E9,9E9]];
            P04W17_Approach := [[0,0,0],[1,0,0,0],[0,0,0,0],[9E9,9E9,9E9,9E9,9E9,9E9]];
            P04W17_Retract := [[0,0,0],[1,0,0,0],[0,0,0,0],[9E9,9E9,9E9,9E9,9E9,9E9]];
            P04W17_Trans := [[0,0,0],[1,0,0,0],[0,0,0,0],[9E9,9E9,9E9,9E9,9E9,9E9]];
        ELSEIF slot = 18 THEN
            P04W18_Used := FALSE;
            P04W18_SubType := 0;
            P04W18_ToolSel := 0;
            P04W18_LenMM := 0;
            P04W18_ArcStart := [[0,0,0],[1,0,0,0],[0,0,0,0],[9E9,9E9,9E9,9E9,9E9,9E9]];
            P04W18_ArcEnd := [[0,0,0],[1,0,0,0],[0,0,0,0],[9E9,9E9,9E9,9E9,9E9,9E9]];
            P04W18_Approach := [[0,0,0],[1,0,0,0],[0,0,0,0],[9E9,9E9,9E9,9E9,9E9,9E9]];
            P04W18_Retract := [[0,0,0],[1,0,0,0],[0,0,0,0],[9E9,9E9,9E9,9E9,9E9,9E9]];
            P04W18_Trans := [[0,0,0],[1,0,0,0],[0,0,0,0],[9E9,9E9,9E9,9E9,9E9,9E9]];
        ELSEIF slot = 19 THEN
            P04W19_Used := FALSE;
            P04W19_SubType := 0;
            P04W19_ToolSel := 0;
            P04W19_LenMM := 0;
            P04W19_ArcStart := [[0,0,0],[1,0,0,0],[0,0,0,0],[9E9,9E9,9E9,9E9,9E9,9E9]];
            P04W19_ArcEnd := [[0,0,0],[1,0,0,0],[0,0,0,0],[9E9,9E9,9E9,9E9,9E9,9E9]];
            P04W19_Approach := [[0,0,0],[1,0,0,0],[0,0,0,0],[9E9,9E9,9E9,9E9,9E9,9E9]];
            P04W19_Retract := [[0,0,0],[1,0,0,0],[0,0,0,0],[9E9,9E9,9E9,9E9,9E9,9E9]];
            P04W19_Trans := [[0,0,0],[1,0,0,0],[0,0,0,0],[9E9,9E9,9E9,9E9,9E9,9E9]];
        ELSEIF slot = 20 THEN
            P04W20_Used := FALSE;
            P04W20_SubType := 0;
            P04W20_ToolSel := 0;
            P04W20_LenMM := 0;
            P04W20_ArcStart := [[0,0,0],[1,0,0,0],[0,0,0,0],[9E9,9E9,9E9,9E9,9E9,9E9]];
            P04W20_ArcEnd := [[0,0,0],[1,0,0,0],[0,0,0,0],[9E9,9E9,9E9,9E9,9E9,9E9]];
            P04W20_Approach := [[0,0,0],[1,0,0,0],[0,0,0,0],[9E9,9E9,9E9,9E9,9E9,9E9]];
            P04W20_Retract := [[0,0,0],[1,0,0,0],[0,0,0,0],[9E9,9E9,9E9,9E9,9E9,9E9]];
            P04W20_Trans := [[0,0,0],[1,0,0,0],[0,0,0,0],[9E9,9E9,9E9,9E9,9E9,9E9]];
        ELSEIF slot = 21 THEN
            P04W21_Used := FALSE;
            P04W21_SubType := 0;
            P04W21_ToolSel := 0;
            P04W21_LenMM := 0;
            P04W21_ArcStart := [[0,0,0],[1,0,0,0],[0,0,0,0],[9E9,9E9,9E9,9E9,9E9,9E9]];
            P04W21_ArcEnd := [[0,0,0],[1,0,0,0],[0,0,0,0],[9E9,9E9,9E9,9E9,9E9,9E9]];
            P04W21_Approach := [[0,0,0],[1,0,0,0],[0,0,0,0],[9E9,9E9,9E9,9E9,9E9,9E9]];
            P04W21_Retract := [[0,0,0],[1,0,0,0],[0,0,0,0],[9E9,9E9,9E9,9E9,9E9,9E9]];
            P04W21_Trans := [[0,0,0],[1,0,0,0],[0,0,0,0],[9E9,9E9,9E9,9E9,9E9,9E9]];
        ELSEIF slot = 22 THEN
            P04W22_Used := FALSE;
            P04W22_SubType := 0;
            P04W22_ToolSel := 0;
            P04W22_LenMM := 0;
            P04W22_ArcStart := [[0,0,0],[1,0,0,0],[0,0,0,0],[9E9,9E9,9E9,9E9,9E9,9E9]];
            P04W22_ArcEnd := [[0,0,0],[1,0,0,0],[0,0,0,0],[9E9,9E9,9E9,9E9,9E9,9E9]];
            P04W22_Approach := [[0,0,0],[1,0,0,0],[0,0,0,0],[9E9,9E9,9E9,9E9,9E9,9E9]];
            P04W22_Retract := [[0,0,0],[1,0,0,0],[0,0,0,0],[9E9,9E9,9E9,9E9,9E9,9E9]];
            P04W22_Trans := [[0,0,0],[1,0,0,0],[0,0,0,0],[9E9,9E9,9E9,9E9,9E9,9E9]];
        ELSEIF slot = 23 THEN
            P04W23_Used := FALSE;
            P04W23_SubType := 0;
            P04W23_ToolSel := 0;
            P04W23_LenMM := 0;
            P04W23_ArcStart := [[0,0,0],[1,0,0,0],[0,0,0,0],[9E9,9E9,9E9,9E9,9E9,9E9]];
            P04W23_ArcEnd := [[0,0,0],[1,0,0,0],[0,0,0,0],[9E9,9E9,9E9,9E9,9E9,9E9]];
            P04W23_Approach := [[0,0,0],[1,0,0,0],[0,0,0,0],[9E9,9E9,9E9,9E9,9E9,9E9]];
            P04W23_Retract := [[0,0,0],[1,0,0,0],[0,0,0,0],[9E9,9E9,9E9,9E9,9E9,9E9]];
            P04W23_Trans := [[0,0,0],[1,0,0,0],[0,0,0,0],[9E9,9E9,9E9,9E9,9E9,9E9]];
        ELSEIF slot = 24 THEN
            P04W24_Used := FALSE;
            P04W24_SubType := 0;
            P04W24_ToolSel := 0;
            P04W24_LenMM := 0;
            P04W24_ArcStart := [[0,0,0],[1,0,0,0],[0,0,0,0],[9E9,9E9,9E9,9E9,9E9,9E9]];
            P04W24_ArcEnd := [[0,0,0],[1,0,0,0],[0,0,0,0],[9E9,9E9,9E9,9E9,9E9,9E9]];
            P04W24_Approach := [[0,0,0],[1,0,0,0],[0,0,0,0],[9E9,9E9,9E9,9E9,9E9,9E9]];
            P04W24_Retract := [[0,0,0],[1,0,0,0],[0,0,0,0],[9E9,9E9,9E9,9E9,9E9,9E9]];
            P04W24_Trans := [[0,0,0],[1,0,0,0],[0,0,0,0],[9E9,9E9,9E9,9E9,9E9,9E9]];
        ELSEIF slot = 25 THEN
            P04W25_Used := FALSE;
            P04W25_SubType := 0;
            P04W25_ToolSel := 0;
            P04W25_LenMM := 0;
            P04W25_ArcStart := [[0,0,0],[1,0,0,0],[0,0,0,0],[9E9,9E9,9E9,9E9,9E9,9E9]];
            P04W25_ArcEnd := [[0,0,0],[1,0,0,0],[0,0,0,0],[9E9,9E9,9E9,9E9,9E9,9E9]];
            P04W25_Approach := [[0,0,0],[1,0,0,0],[0,0,0,0],[9E9,9E9,9E9,9E9,9E9,9E9]];
            P04W25_Retract := [[0,0,0],[1,0,0,0],[0,0,0,0],[9E9,9E9,9E9,9E9,9E9,9E9]];
            P04W25_Trans := [[0,0,0],[1,0,0,0],[0,0,0,0],[9E9,9E9,9E9,9E9,9E9,9E9]];
        ELSEIF slot = 26 THEN
            P04W26_Used := FALSE;
            P04W26_SubType := 0;
            P04W26_ToolSel := 0;
            P04W26_LenMM := 0;
            P04W26_ArcStart := [[0,0,0],[1,0,0,0],[0,0,0,0],[9E9,9E9,9E9,9E9,9E9,9E9]];
            P04W26_ArcEnd := [[0,0,0],[1,0,0,0],[0,0,0,0],[9E9,9E9,9E9,9E9,9E9,9E9]];
            P04W26_Approach := [[0,0,0],[1,0,0,0],[0,0,0,0],[9E9,9E9,9E9,9E9,9E9,9E9]];
            P04W26_Retract := [[0,0,0],[1,0,0,0],[0,0,0,0],[9E9,9E9,9E9,9E9,9E9,9E9]];
            P04W26_Trans := [[0,0,0],[1,0,0,0],[0,0,0,0],[9E9,9E9,9E9,9E9,9E9,9E9]];
        ELSEIF slot = 27 THEN
            P04W27_Used := FALSE;
            P04W27_SubType := 0;
            P04W27_ToolSel := 0;
            P04W27_LenMM := 0;
            P04W27_ArcStart := [[0,0,0],[1,0,0,0],[0,0,0,0],[9E9,9E9,9E9,9E9,9E9,9E9]];
            P04W27_ArcEnd := [[0,0,0],[1,0,0,0],[0,0,0,0],[9E9,9E9,9E9,9E9,9E9,9E9]];
            P04W27_Approach := [[0,0,0],[1,0,0,0],[0,0,0,0],[9E9,9E9,9E9,9E9,9E9,9E9]];
            P04W27_Retract := [[0,0,0],[1,0,0,0],[0,0,0,0],[9E9,9E9,9E9,9E9,9E9,9E9]];
            P04W27_Trans := [[0,0,0],[1,0,0,0],[0,0,0,0],[9E9,9E9,9E9,9E9,9E9,9E9]];
        ELSEIF slot = 28 THEN
            P04W28_Used := FALSE;
            P04W28_SubType := 0;
            P04W28_ToolSel := 0;
            P04W28_LenMM := 0;
            P04W28_ArcStart := [[0,0,0],[1,0,0,0],[0,0,0,0],[9E9,9E9,9E9,9E9,9E9,9E9]];
            P04W28_ArcEnd := [[0,0,0],[1,0,0,0],[0,0,0,0],[9E9,9E9,9E9,9E9,9E9,9E9]];
            P04W28_Approach := [[0,0,0],[1,0,0,0],[0,0,0,0],[9E9,9E9,9E9,9E9,9E9,9E9]];
            P04W28_Retract := [[0,0,0],[1,0,0,0],[0,0,0,0],[9E9,9E9,9E9,9E9,9E9,9E9]];
            P04W28_Trans := [[0,0,0],[1,0,0,0],[0,0,0,0],[9E9,9E9,9E9,9E9,9E9,9E9]];
        ELSEIF slot = 29 THEN
            P04W29_Used := FALSE;
            P04W29_SubType := 0;
            P04W29_ToolSel := 0;
            P04W29_LenMM := 0;
            P04W29_ArcStart := [[0,0,0],[1,0,0,0],[0,0,0,0],[9E9,9E9,9E9,9E9,9E9,9E9]];
            P04W29_ArcEnd := [[0,0,0],[1,0,0,0],[0,0,0,0],[9E9,9E9,9E9,9E9,9E9,9E9]];
            P04W29_Approach := [[0,0,0],[1,0,0,0],[0,0,0,0],[9E9,9E9,9E9,9E9,9E9,9E9]];
            P04W29_Retract := [[0,0,0],[1,0,0,0],[0,0,0,0],[9E9,9E9,9E9,9E9,9E9,9E9]];
            P04W29_Trans := [[0,0,0],[1,0,0,0],[0,0,0,0],[9E9,9E9,9E9,9E9,9E9,9E9]];
        ELSEIF slot = 30 THEN
            P04W30_Used := FALSE;
            P04W30_SubType := 0;
            P04W30_ToolSel := 0;
            P04W30_LenMM := 0;
            P04W30_ArcStart := [[0,0,0],[1,0,0,0],[0,0,0,0],[9E9,9E9,9E9,9E9,9E9,9E9]];
            P04W30_ArcEnd := [[0,0,0],[1,0,0,0],[0,0,0,0],[9E9,9E9,9E9,9E9,9E9,9E9]];
            P04W30_Approach := [[0,0,0],[1,0,0,0],[0,0,0,0],[9E9,9E9,9E9,9E9,9E9,9E9]];
            P04W30_Retract := [[0,0,0],[1,0,0,0],[0,0,0,0],[9E9,9E9,9E9,9E9,9E9,9E9]];
            P04W30_Trans := [[0,0,0],[1,0,0,0],[0,0,0,0],[9E9,9E9,9E9,9E9,9E9,9E9]];
        ELSE
            TPWrite "Invalid weld slot.";
        ENDIF
    ENDPROC

    PROC StoreNextFree_P04(num subType, num toolSel, num lenMM,
                       robtarget arcStart, robtarget arcEnd, robtarget approach, robtarget retract, robtarget trans)
        IF NOT P04W01_Used THEN
            StoreSlot_P04 1, subType, toolSel, lenMM, arcStart, arcEnd, approach, retract, trans;
            nWeldsP04 := nWeldsP04 + 1;
            RETURN;
        ELSEIF NOT P04W02_Used THEN
            StoreSlot_P04 2, subType, toolSel, lenMM, arcStart, arcEnd, approach, retract, trans;
            nWeldsP04 := nWeldsP04 + 1;
            RETURN;
        ELSEIF NOT P04W03_Used THEN
            StoreSlot_P04 3, subType, toolSel, lenMM, arcStart, arcEnd, approach, retract, trans;
            nWeldsP04 := nWeldsP04 + 1;
            RETURN;
        ELSEIF NOT P04W04_Used THEN
            StoreSlot_P04 4, subType, toolSel, lenMM, arcStart, arcEnd, approach, retract, trans;
            nWeldsP04 := nWeldsP04 + 1;
            RETURN;
        ELSEIF NOT P04W05_Used THEN
            StoreSlot_P04 5, subType, toolSel, lenMM, arcStart, arcEnd, approach, retract, trans;
            nWeldsP04 := nWeldsP04 + 1;
            RETURN;
        ELSEIF NOT P04W06_Used THEN
            StoreSlot_P04 6, subType, toolSel, lenMM, arcStart, arcEnd, approach, retract, trans;
            nWeldsP04 := nWeldsP04 + 1;
            RETURN;
        ELSEIF NOT P04W07_Used THEN
            StoreSlot_P04 7, subType, toolSel, lenMM, arcStart, arcEnd, approach, retract, trans;
            nWeldsP04 := nWeldsP04 + 1;
            RETURN;
        ELSEIF NOT P04W08_Used THEN
            StoreSlot_P04 8, subType, toolSel, lenMM, arcStart, arcEnd, approach, retract, trans;
            nWeldsP04 := nWeldsP04 + 1;
            RETURN;
        ELSEIF NOT P04W09_Used THEN
            StoreSlot_P04 9, subType, toolSel, lenMM, arcStart, arcEnd, approach, retract, trans;
            nWeldsP04 := nWeldsP04 + 1;
            RETURN;
        ELSEIF NOT P04W10_Used THEN
            StoreSlot_P04 10, subType, toolSel, lenMM, arcStart, arcEnd, approach, retract, trans;
            nWeldsP04 := nWeldsP04 + 1;
            RETURN;
        ELSEIF NOT P04W11_Used THEN
            StoreSlot_P04 11, subType, toolSel, lenMM, arcStart, arcEnd, approach, retract, trans;
            nWeldsP04 := nWeldsP04 + 1;
            RETURN;
        ELSEIF NOT P04W12_Used THEN
            StoreSlot_P04 12, subType, toolSel, lenMM, arcStart, arcEnd, approach, retract, trans;
            nWeldsP04 := nWeldsP04 + 1;
            RETURN;
        ELSEIF NOT P04W13_Used THEN
            StoreSlot_P04 13, subType, toolSel, lenMM, arcStart, arcEnd, approach, retract, trans;
            nWeldsP04 := nWeldsP04 + 1;
            RETURN;
        ELSEIF NOT P04W14_Used THEN
            StoreSlot_P04 14, subType, toolSel, lenMM, arcStart, arcEnd, approach, retract, trans;
            nWeldsP04 := nWeldsP04 + 1;
            RETURN;
        ELSEIF NOT P04W15_Used THEN
            StoreSlot_P04 15, subType, toolSel, lenMM, arcStart, arcEnd, approach, retract, trans;
            nWeldsP04 := nWeldsP04 + 1;
            RETURN;
        ELSEIF NOT P04W16_Used THEN
            StoreSlot_P04 16, subType, toolSel, lenMM, arcStart, arcEnd, approach, retract, trans;
            nWeldsP04 := nWeldsP04 + 1;
            RETURN;
        ELSEIF NOT P04W17_Used THEN
            StoreSlot_P04 17, subType, toolSel, lenMM, arcStart, arcEnd, approach, retract, trans;
            nWeldsP04 := nWeldsP04 + 1;
            RETURN;
        ELSEIF NOT P04W18_Used THEN
            StoreSlot_P04 18, subType, toolSel, lenMM, arcStart, arcEnd, approach, retract, trans;
            nWeldsP04 := nWeldsP04 + 1;
            RETURN;
        ELSEIF NOT P04W19_Used THEN
            StoreSlot_P04 19, subType, toolSel, lenMM, arcStart, arcEnd, approach, retract, trans;
            nWeldsP04 := nWeldsP04 + 1;
            RETURN;
        ELSEIF NOT P04W20_Used THEN
            StoreSlot_P04 20, subType, toolSel, lenMM, arcStart, arcEnd, approach, retract, trans;
            nWeldsP04 := nWeldsP04 + 1;
            RETURN;
        ELSEIF NOT P04W21_Used THEN
            StoreSlot_P04 21, subType, toolSel, lenMM, arcStart, arcEnd, approach, retract, trans;
            nWeldsP04 := nWeldsP04 + 1;
            RETURN;
        ELSEIF NOT P04W22_Used THEN
            StoreSlot_P04 22, subType, toolSel, lenMM, arcStart, arcEnd, approach, retract, trans;
            nWeldsP04 := nWeldsP04 + 1;
            RETURN;
        ELSEIF NOT P04W23_Used THEN
            StoreSlot_P04 23, subType, toolSel, lenMM, arcStart, arcEnd, approach, retract, trans;
            nWeldsP04 := nWeldsP04 + 1;
            RETURN;
        ELSEIF NOT P04W24_Used THEN
            StoreSlot_P04 24, subType, toolSel, lenMM, arcStart, arcEnd, approach, retract, trans;
            nWeldsP04 := nWeldsP04 + 1;
            RETURN;
        ELSEIF NOT P04W25_Used THEN
            StoreSlot_P04 25, subType, toolSel, lenMM, arcStart, arcEnd, approach, retract, trans;
            nWeldsP04 := nWeldsP04 + 1;
            RETURN;
        ELSEIF NOT P04W26_Used THEN
            StoreSlot_P04 26, subType, toolSel, lenMM, arcStart, arcEnd, approach, retract, trans;
            nWeldsP04 := nWeldsP04 + 1;
            RETURN;
        ELSEIF NOT P04W27_Used THEN
            StoreSlot_P04 27, subType, toolSel, lenMM, arcStart, arcEnd, approach, retract, trans;
            nWeldsP04 := nWeldsP04 + 1;
            RETURN;
        ELSEIF NOT P04W28_Used THEN
            StoreSlot_P04 28, subType, toolSel, lenMM, arcStart, arcEnd, approach, retract, trans;
            nWeldsP04 := nWeldsP04 + 1;
            RETURN;
        ELSEIF NOT P04W29_Used THEN
            StoreSlot_P04 29, subType, toolSel, lenMM, arcStart, arcEnd, approach, retract, trans;
            nWeldsP04 := nWeldsP04 + 1;
            RETURN;
        ELSEIF NOT P04W30_Used THEN
            StoreSlot_P04 30, subType, toolSel, lenMM, arcStart, arcEnd, approach, retract, trans;
            nWeldsP04 := nWeldsP04 + 1;
            RETURN;
        ELSE
            TPWrite "No free weld slots available.";
        ENDIF
    ENDPROC

    PROC StoreSlot_P05(num slot, num subType, num toolSel, num lenMM,
                       robtarget arcStart, robtarget arcEnd, robtarget approach, robtarget retract, robtarget trans)
        IF slot = 1 THEN
            P05W01_SubType := subType;
            P05W01_ToolSel := toolSel;
            P05W01_LenMM := lenMM;
            P05W01_ArcStart := arcStart;
            P05W01_ArcEnd := arcEnd;
            P05W01_Approach := approach;
            P05W01_Retract := retract;
            P05W01_Trans := trans;
            P05W01_Used := TRUE;
        ELSEIF slot = 2 THEN
            P05W02_SubType := subType;
            P05W02_ToolSel := toolSel;
            P05W02_LenMM := lenMM;
            P05W02_ArcStart := arcStart;
            P05W02_ArcEnd := arcEnd;
            P05W02_Approach := approach;
            P05W02_Retract := retract;
            P05W02_Trans := trans;
            P05W02_Used := TRUE;
        ELSEIF slot = 3 THEN
            P05W03_SubType := subType;
            P05W03_ToolSel := toolSel;
            P05W03_LenMM := lenMM;
            P05W03_ArcStart := arcStart;
            P05W03_ArcEnd := arcEnd;
            P05W03_Approach := approach;
            P05W03_Retract := retract;
            P05W03_Trans := trans;
            P05W03_Used := TRUE;
        ELSEIF slot = 4 THEN
            P05W04_SubType := subType;
            P05W04_ToolSel := toolSel;
            P05W04_LenMM := lenMM;
            P05W04_ArcStart := arcStart;
            P05W04_ArcEnd := arcEnd;
            P05W04_Approach := approach;
            P05W04_Retract := retract;
            P05W04_Trans := trans;
            P05W04_Used := TRUE;
        ELSEIF slot = 5 THEN
            P05W05_SubType := subType;
            P05W05_ToolSel := toolSel;
            P05W05_LenMM := lenMM;
            P05W05_ArcStart := arcStart;
            P05W05_ArcEnd := arcEnd;
            P05W05_Approach := approach;
            P05W05_Retract := retract;
            P05W05_Trans := trans;
            P05W05_Used := TRUE;
        ELSEIF slot = 6 THEN
            P05W06_SubType := subType;
            P05W06_ToolSel := toolSel;
            P05W06_LenMM := lenMM;
            P05W06_ArcStart := arcStart;
            P05W06_ArcEnd := arcEnd;
            P05W06_Approach := approach;
            P05W06_Retract := retract;
            P05W06_Trans := trans;
            P05W06_Used := TRUE;
        ELSEIF slot = 7 THEN
            P05W07_SubType := subType;
            P05W07_ToolSel := toolSel;
            P05W07_LenMM := lenMM;
            P05W07_ArcStart := arcStart;
            P05W07_ArcEnd := arcEnd;
            P05W07_Approach := approach;
            P05W07_Retract := retract;
            P05W07_Trans := trans;
            P05W07_Used := TRUE;
        ELSEIF slot = 8 THEN
            P05W08_SubType := subType;
            P05W08_ToolSel := toolSel;
            P05W08_LenMM := lenMM;
            P05W08_ArcStart := arcStart;
            P05W08_ArcEnd := arcEnd;
            P05W08_Approach := approach;
            P05W08_Retract := retract;
            P05W08_Trans := trans;
            P05W08_Used := TRUE;
        ELSEIF slot = 9 THEN
            P05W09_SubType := subType;
            P05W09_ToolSel := toolSel;
            P05W09_LenMM := lenMM;
            P05W09_ArcStart := arcStart;
            P05W09_ArcEnd := arcEnd;
            P05W09_Approach := approach;
            P05W09_Retract := retract;
            P05W09_Trans := trans;
            P05W09_Used := TRUE;
        ELSEIF slot = 10 THEN
            P05W10_SubType := subType;
            P05W10_ToolSel := toolSel;
            P05W10_LenMM := lenMM;
            P05W10_ArcStart := arcStart;
            P05W10_ArcEnd := arcEnd;
            P05W10_Approach := approach;
            P05W10_Retract := retract;
            P05W10_Trans := trans;
            P05W10_Used := TRUE;
        ELSEIF slot = 11 THEN
            P05W11_SubType := subType;
            P05W11_ToolSel := toolSel;
            P05W11_LenMM := lenMM;
            P05W11_ArcStart := arcStart;
            P05W11_ArcEnd := arcEnd;
            P05W11_Approach := approach;
            P05W11_Retract := retract;
            P05W11_Trans := trans;
            P05W11_Used := TRUE;
        ELSEIF slot = 12 THEN
            P05W12_SubType := subType;
            P05W12_ToolSel := toolSel;
            P05W12_LenMM := lenMM;
            P05W12_ArcStart := arcStart;
            P05W12_ArcEnd := arcEnd;
            P05W12_Approach := approach;
            P05W12_Retract := retract;
            P05W12_Trans := trans;
            P05W12_Used := TRUE;
        ELSEIF slot = 13 THEN
            P05W13_SubType := subType;
            P05W13_ToolSel := toolSel;
            P05W13_LenMM := lenMM;
            P05W13_ArcStart := arcStart;
            P05W13_ArcEnd := arcEnd;
            P05W13_Approach := approach;
            P05W13_Retract := retract;
            P05W13_Trans := trans;
            P05W13_Used := TRUE;
        ELSEIF slot = 14 THEN
            P05W14_SubType := subType;
            P05W14_ToolSel := toolSel;
            P05W14_LenMM := lenMM;
            P05W14_ArcStart := arcStart;
            P05W14_ArcEnd := arcEnd;
            P05W14_Approach := approach;
            P05W14_Retract := retract;
            P05W14_Trans := trans;
            P05W14_Used := TRUE;
        ELSEIF slot = 15 THEN
            P05W15_SubType := subType;
            P05W15_ToolSel := toolSel;
            P05W15_LenMM := lenMM;
            P05W15_ArcStart := arcStart;
            P05W15_ArcEnd := arcEnd;
            P05W15_Approach := approach;
            P05W15_Retract := retract;
            P05W15_Trans := trans;
            P05W15_Used := TRUE;
        ELSEIF slot = 16 THEN
            P05W16_SubType := subType;
            P05W16_ToolSel := toolSel;
            P05W16_LenMM := lenMM;
            P05W16_ArcStart := arcStart;
            P05W16_ArcEnd := arcEnd;
            P05W16_Approach := approach;
            P05W16_Retract := retract;
            P05W16_Trans := trans;
            P05W16_Used := TRUE;
        ELSEIF slot = 17 THEN
            P05W17_SubType := subType;
            P05W17_ToolSel := toolSel;
            P05W17_LenMM := lenMM;
            P05W17_ArcStart := arcStart;
            P05W17_ArcEnd := arcEnd;
            P05W17_Approach := approach;
            P05W17_Retract := retract;
            P05W17_Trans := trans;
            P05W17_Used := TRUE;
        ELSEIF slot = 18 THEN
            P05W18_SubType := subType;
            P05W18_ToolSel := toolSel;
            P05W18_LenMM := lenMM;
            P05W18_ArcStart := arcStart;
            P05W18_ArcEnd := arcEnd;
            P05W18_Approach := approach;
            P05W18_Retract := retract;
            P05W18_Trans := trans;
            P05W18_Used := TRUE;
        ELSEIF slot = 19 THEN
            P05W19_SubType := subType;
            P05W19_ToolSel := toolSel;
            P05W19_LenMM := lenMM;
            P05W19_ArcStart := arcStart;
            P05W19_ArcEnd := arcEnd;
            P05W19_Approach := approach;
            P05W19_Retract := retract;
            P05W19_Trans := trans;
            P05W19_Used := TRUE;
        ELSEIF slot = 20 THEN
            P05W20_SubType := subType;
            P05W20_ToolSel := toolSel;
            P05W20_LenMM := lenMM;
            P05W20_ArcStart := arcStart;
            P05W20_ArcEnd := arcEnd;
            P05W20_Approach := approach;
            P05W20_Retract := retract;
            P05W20_Trans := trans;
            P05W20_Used := TRUE;
        ELSEIF slot = 21 THEN
            P05W21_SubType := subType;
            P05W21_ToolSel := toolSel;
            P05W21_LenMM := lenMM;
            P05W21_ArcStart := arcStart;
            P05W21_ArcEnd := arcEnd;
            P05W21_Approach := approach;
            P05W21_Retract := retract;
            P05W21_Trans := trans;
            P05W21_Used := TRUE;
        ELSEIF slot = 22 THEN
            P05W22_SubType := subType;
            P05W22_ToolSel := toolSel;
            P05W22_LenMM := lenMM;
            P05W22_ArcStart := arcStart;
            P05W22_ArcEnd := arcEnd;
            P05W22_Approach := approach;
            P05W22_Retract := retract;
            P05W22_Trans := trans;
            P05W22_Used := TRUE;
        ELSEIF slot = 23 THEN
            P05W23_SubType := subType;
            P05W23_ToolSel := toolSel;
            P05W23_LenMM := lenMM;
            P05W23_ArcStart := arcStart;
            P05W23_ArcEnd := arcEnd;
            P05W23_Approach := approach;
            P05W23_Retract := retract;
            P05W23_Trans := trans;
            P05W23_Used := TRUE;
        ELSEIF slot = 24 THEN
            P05W24_SubType := subType;
            P05W24_ToolSel := toolSel;
            P05W24_LenMM := lenMM;
            P05W24_ArcStart := arcStart;
            P05W24_ArcEnd := arcEnd;
            P05W24_Approach := approach;
            P05W24_Retract := retract;
            P05W24_Trans := trans;
            P05W24_Used := TRUE;
        ELSEIF slot = 25 THEN
            P05W25_SubType := subType;
            P05W25_ToolSel := toolSel;
            P05W25_LenMM := lenMM;
            P05W25_ArcStart := arcStart;
            P05W25_ArcEnd := arcEnd;
            P05W25_Approach := approach;
            P05W25_Retract := retract;
            P05W25_Trans := trans;
            P05W25_Used := TRUE;
        ELSEIF slot = 26 THEN
            P05W26_SubType := subType;
            P05W26_ToolSel := toolSel;
            P05W26_LenMM := lenMM;
            P05W26_ArcStart := arcStart;
            P05W26_ArcEnd := arcEnd;
            P05W26_Approach := approach;
            P05W26_Retract := retract;
            P05W26_Trans := trans;
            P05W26_Used := TRUE;
        ELSEIF slot = 27 THEN
            P05W27_SubType := subType;
            P05W27_ToolSel := toolSel;
            P05W27_LenMM := lenMM;
            P05W27_ArcStart := arcStart;
            P05W27_ArcEnd := arcEnd;
            P05W27_Approach := approach;
            P05W27_Retract := retract;
            P05W27_Trans := trans;
            P05W27_Used := TRUE;
        ELSEIF slot = 28 THEN
            P05W28_SubType := subType;
            P05W28_ToolSel := toolSel;
            P05W28_LenMM := lenMM;
            P05W28_ArcStart := arcStart;
            P05W28_ArcEnd := arcEnd;
            P05W28_Approach := approach;
            P05W28_Retract := retract;
            P05W28_Trans := trans;
            P05W28_Used := TRUE;
        ELSEIF slot = 29 THEN
            P05W29_SubType := subType;
            P05W29_ToolSel := toolSel;
            P05W29_LenMM := lenMM;
            P05W29_ArcStart := arcStart;
            P05W29_ArcEnd := arcEnd;
            P05W29_Approach := approach;
            P05W29_Retract := retract;
            P05W29_Trans := trans;
            P05W29_Used := TRUE;
        ELSEIF slot = 30 THEN
            P05W30_SubType := subType;
            P05W30_ToolSel := toolSel;
            P05W30_LenMM := lenMM;
            P05W30_ArcStart := arcStart;
            P05W30_ArcEnd := arcEnd;
            P05W30_Approach := approach;
            P05W30_Retract := retract;
            P05W30_Trans := trans;
            P05W30_Used := TRUE;
        ELSE
            TPWrite "Invalid weld slot.";
        ENDIF
    ENDPROC

    PROC LoadSlot_P05(num slot, VAR bool used, VAR num subType, VAR num toolSel, VAR num lenMM,
                       VAR robtarget arcStart, VAR robtarget arcEnd, VAR robtarget approach, VAR robtarget retract, VAR robtarget trans)
        IF slot = 1 THEN
            used := P05W01_Used;
            subType := P05W01_SubType;
            toolSel := P05W01_ToolSel;
            lenMM := P05W01_LenMM;
            arcStart := P05W01_ArcStart;
            arcEnd := P05W01_ArcEnd;
            approach := P05W01_Approach;
            retract := P05W01_Retract;
            trans := P05W01_Trans;
        ELSEIF slot = 2 THEN
            used := P05W02_Used;
            subType := P05W02_SubType;
            toolSel := P05W02_ToolSel;
            lenMM := P05W02_LenMM;
            arcStart := P05W02_ArcStart;
            arcEnd := P05W02_ArcEnd;
            approach := P05W02_Approach;
            retract := P05W02_Retract;
            trans := P05W02_Trans;
        ELSEIF slot = 3 THEN
            used := P05W03_Used;
            subType := P05W03_SubType;
            toolSel := P05W03_ToolSel;
            lenMM := P05W03_LenMM;
            arcStart := P05W03_ArcStart;
            arcEnd := P05W03_ArcEnd;
            approach := P05W03_Approach;
            retract := P05W03_Retract;
            trans := P05W03_Trans;
        ELSEIF slot = 4 THEN
            used := P05W04_Used;
            subType := P05W04_SubType;
            toolSel := P05W04_ToolSel;
            lenMM := P05W04_LenMM;
            arcStart := P05W04_ArcStart;
            arcEnd := P05W04_ArcEnd;
            approach := P05W04_Approach;
            retract := P05W04_Retract;
            trans := P05W04_Trans;
        ELSEIF slot = 5 THEN
            used := P05W05_Used;
            subType := P05W05_SubType;
            toolSel := P05W05_ToolSel;
            lenMM := P05W05_LenMM;
            arcStart := P05W05_ArcStart;
            arcEnd := P05W05_ArcEnd;
            approach := P05W05_Approach;
            retract := P05W05_Retract;
            trans := P05W05_Trans;
        ELSEIF slot = 6 THEN
            used := P05W06_Used;
            subType := P05W06_SubType;
            toolSel := P05W06_ToolSel;
            lenMM := P05W06_LenMM;
            arcStart := P05W06_ArcStart;
            arcEnd := P05W06_ArcEnd;
            approach := P05W06_Approach;
            retract := P05W06_Retract;
            trans := P05W06_Trans;
        ELSEIF slot = 7 THEN
            used := P05W07_Used;
            subType := P05W07_SubType;
            toolSel := P05W07_ToolSel;
            lenMM := P05W07_LenMM;
            arcStart := P05W07_ArcStart;
            arcEnd := P05W07_ArcEnd;
            approach := P05W07_Approach;
            retract := P05W07_Retract;
            trans := P05W07_Trans;
        ELSEIF slot = 8 THEN
            used := P05W08_Used;
            subType := P05W08_SubType;
            toolSel := P05W08_ToolSel;
            lenMM := P05W08_LenMM;
            arcStart := P05W08_ArcStart;
            arcEnd := P05W08_ArcEnd;
            approach := P05W08_Approach;
            retract := P05W08_Retract;
            trans := P05W08_Trans;
        ELSEIF slot = 9 THEN
            used := P05W09_Used;
            subType := P05W09_SubType;
            toolSel := P05W09_ToolSel;
            lenMM := P05W09_LenMM;
            arcStart := P05W09_ArcStart;
            arcEnd := P05W09_ArcEnd;
            approach := P05W09_Approach;
            retract := P05W09_Retract;
            trans := P05W09_Trans;
        ELSEIF slot = 10 THEN
            used := P05W10_Used;
            subType := P05W10_SubType;
            toolSel := P05W10_ToolSel;
            lenMM := P05W10_LenMM;
            arcStart := P05W10_ArcStart;
            arcEnd := P05W10_ArcEnd;
            approach := P05W10_Approach;
            retract := P05W10_Retract;
            trans := P05W10_Trans;
        ELSEIF slot = 11 THEN
            used := P05W11_Used;
            subType := P05W11_SubType;
            toolSel := P05W11_ToolSel;
            lenMM := P05W11_LenMM;
            arcStart := P05W11_ArcStart;
            arcEnd := P05W11_ArcEnd;
            approach := P05W11_Approach;
            retract := P05W11_Retract;
            trans := P05W11_Trans;
        ELSEIF slot = 12 THEN
            used := P05W12_Used;
            subType := P05W12_SubType;
            toolSel := P05W12_ToolSel;
            lenMM := P05W12_LenMM;
            arcStart := P05W12_ArcStart;
            arcEnd := P05W12_ArcEnd;
            approach := P05W12_Approach;
            retract := P05W12_Retract;
            trans := P05W12_Trans;
        ELSEIF slot = 13 THEN
            used := P05W13_Used;
            subType := P05W13_SubType;
            toolSel := P05W13_ToolSel;
            lenMM := P05W13_LenMM;
            arcStart := P05W13_ArcStart;
            arcEnd := P05W13_ArcEnd;
            approach := P05W13_Approach;
            retract := P05W13_Retract;
            trans := P05W13_Trans;
        ELSEIF slot = 14 THEN
            used := P05W14_Used;
            subType := P05W14_SubType;
            toolSel := P05W14_ToolSel;
            lenMM := P05W14_LenMM;
            arcStart := P05W14_ArcStart;
            arcEnd := P05W14_ArcEnd;
            approach := P05W14_Approach;
            retract := P05W14_Retract;
            trans := P05W14_Trans;
        ELSEIF slot = 15 THEN
            used := P05W15_Used;
            subType := P05W15_SubType;
            toolSel := P05W15_ToolSel;
            lenMM := P05W15_LenMM;
            arcStart := P05W15_ArcStart;
            arcEnd := P05W15_ArcEnd;
            approach := P05W15_Approach;
            retract := P05W15_Retract;
            trans := P05W15_Trans;
        ELSEIF slot = 16 THEN
            used := P05W16_Used;
            subType := P05W16_SubType;
            toolSel := P05W16_ToolSel;
            lenMM := P05W16_LenMM;
            arcStart := P05W16_ArcStart;
            arcEnd := P05W16_ArcEnd;
            approach := P05W16_Approach;
            retract := P05W16_Retract;
            trans := P05W16_Trans;
        ELSEIF slot = 17 THEN
            used := P05W17_Used;
            subType := P05W17_SubType;
            toolSel := P05W17_ToolSel;
            lenMM := P05W17_LenMM;
            arcStart := P05W17_ArcStart;
            arcEnd := P05W17_ArcEnd;
            approach := P05W17_Approach;
            retract := P05W17_Retract;
            trans := P05W17_Trans;
        ELSEIF slot = 18 THEN
            used := P05W18_Used;
            subType := P05W18_SubType;
            toolSel := P05W18_ToolSel;
            lenMM := P05W18_LenMM;
            arcStart := P05W18_ArcStart;
            arcEnd := P05W18_ArcEnd;
            approach := P05W18_Approach;
            retract := P05W18_Retract;
            trans := P05W18_Trans;
        ELSEIF slot = 19 THEN
            used := P05W19_Used;
            subType := P05W19_SubType;
            toolSel := P05W19_ToolSel;
            lenMM := P05W19_LenMM;
            arcStart := P05W19_ArcStart;
            arcEnd := P05W19_ArcEnd;
            approach := P05W19_Approach;
            retract := P05W19_Retract;
            trans := P05W19_Trans;
        ELSEIF slot = 20 THEN
            used := P05W20_Used;
            subType := P05W20_SubType;
            toolSel := P05W20_ToolSel;
            lenMM := P05W20_LenMM;
            arcStart := P05W20_ArcStart;
            arcEnd := P05W20_ArcEnd;
            approach := P05W20_Approach;
            retract := P05W20_Retract;
            trans := P05W20_Trans;
        ELSEIF slot = 21 THEN
            used := P05W21_Used;
            subType := P05W21_SubType;
            toolSel := P05W21_ToolSel;
            lenMM := P05W21_LenMM;
            arcStart := P05W21_ArcStart;
            arcEnd := P05W21_ArcEnd;
            approach := P05W21_Approach;
            retract := P05W21_Retract;
            trans := P05W21_Trans;
        ELSEIF slot = 22 THEN
            used := P05W22_Used;
            subType := P05W22_SubType;
            toolSel := P05W22_ToolSel;
            lenMM := P05W22_LenMM;
            arcStart := P05W22_ArcStart;
            arcEnd := P05W22_ArcEnd;
            approach := P05W22_Approach;
            retract := P05W22_Retract;
            trans := P05W22_Trans;
        ELSEIF slot = 23 THEN
            used := P05W23_Used;
            subType := P05W23_SubType;
            toolSel := P05W23_ToolSel;
            lenMM := P05W23_LenMM;
            arcStart := P05W23_ArcStart;
            arcEnd := P05W23_ArcEnd;
            approach := P05W23_Approach;
            retract := P05W23_Retract;
            trans := P05W23_Trans;
        ELSEIF slot = 24 THEN
            used := P05W24_Used;
            subType := P05W24_SubType;
            toolSel := P05W24_ToolSel;
            lenMM := P05W24_LenMM;
            arcStart := P05W24_ArcStart;
            arcEnd := P05W24_ArcEnd;
            approach := P05W24_Approach;
            retract := P05W24_Retract;
            trans := P05W24_Trans;
        ELSEIF slot = 25 THEN
            used := P05W25_Used;
            subType := P05W25_SubType;
            toolSel := P05W25_ToolSel;
            lenMM := P05W25_LenMM;
            arcStart := P05W25_ArcStart;
            arcEnd := P05W25_ArcEnd;
            approach := P05W25_Approach;
            retract := P05W25_Retract;
            trans := P05W25_Trans;
        ELSEIF slot = 26 THEN
            used := P05W26_Used;
            subType := P05W26_SubType;
            toolSel := P05W26_ToolSel;
            lenMM := P05W26_LenMM;
            arcStart := P05W26_ArcStart;
            arcEnd := P05W26_ArcEnd;
            approach := P05W26_Approach;
            retract := P05W26_Retract;
            trans := P05W26_Trans;
        ELSEIF slot = 27 THEN
            used := P05W27_Used;
            subType := P05W27_SubType;
            toolSel := P05W27_ToolSel;
            lenMM := P05W27_LenMM;
            arcStart := P05W27_ArcStart;
            arcEnd := P05W27_ArcEnd;
            approach := P05W27_Approach;
            retract := P05W27_Retract;
            trans := P05W27_Trans;
        ELSEIF slot = 28 THEN
            used := P05W28_Used;
            subType := P05W28_SubType;
            toolSel := P05W28_ToolSel;
            lenMM := P05W28_LenMM;
            arcStart := P05W28_ArcStart;
            arcEnd := P05W28_ArcEnd;
            approach := P05W28_Approach;
            retract := P05W28_Retract;
            trans := P05W28_Trans;
        ELSEIF slot = 29 THEN
            used := P05W29_Used;
            subType := P05W29_SubType;
            toolSel := P05W29_ToolSel;
            lenMM := P05W29_LenMM;
            arcStart := P05W29_ArcStart;
            arcEnd := P05W29_ArcEnd;
            approach := P05W29_Approach;
            retract := P05W29_Retract;
            trans := P05W29_Trans;
        ELSEIF slot = 30 THEN
            used := P05W30_Used;
            subType := P05W30_SubType;
            toolSel := P05W30_ToolSel;
            lenMM := P05W30_LenMM;
            arcStart := P05W30_ArcStart;
            arcEnd := P05W30_ArcEnd;
            approach := P05W30_Approach;
            retract := P05W30_Retract;
            trans := P05W30_Trans;
        ELSE
            used := FALSE;
        ENDIF
    ENDPROC

    PROC ClearSlot_P05(num slot)
        IF slot = 1 THEN
            P05W01_Used := FALSE;
            P05W01_SubType := 0;
            P05W01_ToolSel := 0;
            P05W01_LenMM := 0;
            P05W01_ArcStart := [[0,0,0],[1,0,0,0],[0,0,0,0],[9E9,9E9,9E9,9E9,9E9,9E9]];
            P05W01_ArcEnd := [[0,0,0],[1,0,0,0],[0,0,0,0],[9E9,9E9,9E9,9E9,9E9,9E9]];
            P05W01_Approach := [[0,0,0],[1,0,0,0],[0,0,0,0],[9E9,9E9,9E9,9E9,9E9,9E9]];
            P05W01_Retract := [[0,0,0],[1,0,0,0],[0,0,0,0],[9E9,9E9,9E9,9E9,9E9,9E9]];
            P05W01_Trans := [[0,0,0],[1,0,0,0],[0,0,0,0],[9E9,9E9,9E9,9E9,9E9,9E9]];
        ELSEIF slot = 2 THEN
            P05W02_Used := FALSE;
            P05W02_SubType := 0;
            P05W02_ToolSel := 0;
            P05W02_LenMM := 0;
            P05W02_ArcStart := [[0,0,0],[1,0,0,0],[0,0,0,0],[9E9,9E9,9E9,9E9,9E9,9E9]];
            P05W02_ArcEnd := [[0,0,0],[1,0,0,0],[0,0,0,0],[9E9,9E9,9E9,9E9,9E9,9E9]];
            P05W02_Approach := [[0,0,0],[1,0,0,0],[0,0,0,0],[9E9,9E9,9E9,9E9,9E9,9E9]];
            P05W02_Retract := [[0,0,0],[1,0,0,0],[0,0,0,0],[9E9,9E9,9E9,9E9,9E9,9E9]];
            P05W02_Trans := [[0,0,0],[1,0,0,0],[0,0,0,0],[9E9,9E9,9E9,9E9,9E9,9E9]];
        ELSEIF slot = 3 THEN
            P05W03_Used := FALSE;
            P05W03_SubType := 0;
            P05W03_ToolSel := 0;
            P05W03_LenMM := 0;
            P05W03_ArcStart := [[0,0,0],[1,0,0,0],[0,0,0,0],[9E9,9E9,9E9,9E9,9E9,9E9]];
            P05W03_ArcEnd := [[0,0,0],[1,0,0,0],[0,0,0,0],[9E9,9E9,9E9,9E9,9E9,9E9]];
            P05W03_Approach := [[0,0,0],[1,0,0,0],[0,0,0,0],[9E9,9E9,9E9,9E9,9E9,9E9]];
            P05W03_Retract := [[0,0,0],[1,0,0,0],[0,0,0,0],[9E9,9E9,9E9,9E9,9E9,9E9]];
            P05W03_Trans := [[0,0,0],[1,0,0,0],[0,0,0,0],[9E9,9E9,9E9,9E9,9E9,9E9]];
        ELSEIF slot = 4 THEN
            P05W04_Used := FALSE;
            P05W04_SubType := 0;
            P05W04_ToolSel := 0;
            P05W04_LenMM := 0;
            P05W04_ArcStart := [[0,0,0],[1,0,0,0],[0,0,0,0],[9E9,9E9,9E9,9E9,9E9,9E9]];
            P05W04_ArcEnd := [[0,0,0],[1,0,0,0],[0,0,0,0],[9E9,9E9,9E9,9E9,9E9,9E9]];
            P05W04_Approach := [[0,0,0],[1,0,0,0],[0,0,0,0],[9E9,9E9,9E9,9E9,9E9,9E9]];
            P05W04_Retract := [[0,0,0],[1,0,0,0],[0,0,0,0],[9E9,9E9,9E9,9E9,9E9,9E9]];
            P05W04_Trans := [[0,0,0],[1,0,0,0],[0,0,0,0],[9E9,9E9,9E9,9E9,9E9,9E9]];
        ELSEIF slot = 5 THEN
            P05W05_Used := FALSE;
            P05W05_SubType := 0;
            P05W05_ToolSel := 0;
            P05W05_LenMM := 0;
            P05W05_ArcStart := [[0,0,0],[1,0,0,0],[0,0,0,0],[9E9,9E9,9E9,9E9,9E9,9E9]];
            P05W05_ArcEnd := [[0,0,0],[1,0,0,0],[0,0,0,0],[9E9,9E9,9E9,9E9,9E9,9E9]];
            P05W05_Approach := [[0,0,0],[1,0,0,0],[0,0,0,0],[9E9,9E9,9E9,9E9,9E9,9E9]];
            P05W05_Retract := [[0,0,0],[1,0,0,0],[0,0,0,0],[9E9,9E9,9E9,9E9,9E9,9E9]];
            P05W05_Trans := [[0,0,0],[1,0,0,0],[0,0,0,0],[9E9,9E9,9E9,9E9,9E9,9E9]];
        ELSEIF slot = 6 THEN
            P05W06_Used := FALSE;
            P05W06_SubType := 0;
            P05W06_ToolSel := 0;
            P05W06_LenMM := 0;
            P05W06_ArcStart := [[0,0,0],[1,0,0,0],[0,0,0,0],[9E9,9E9,9E9,9E9,9E9,9E9]];
            P05W06_ArcEnd := [[0,0,0],[1,0,0,0],[0,0,0,0],[9E9,9E9,9E9,9E9,9E9,9E9]];
            P05W06_Approach := [[0,0,0],[1,0,0,0],[0,0,0,0],[9E9,9E9,9E9,9E9,9E9,9E9]];
            P05W06_Retract := [[0,0,0],[1,0,0,0],[0,0,0,0],[9E9,9E9,9E9,9E9,9E9,9E9]];
            P05W06_Trans := [[0,0,0],[1,0,0,0],[0,0,0,0],[9E9,9E9,9E9,9E9,9E9,9E9]];
        ELSEIF slot = 7 THEN
            P05W07_Used := FALSE;
            P05W07_SubType := 0;
            P05W07_ToolSel := 0;
            P05W07_LenMM := 0;
            P05W07_ArcStart := [[0,0,0],[1,0,0,0],[0,0,0,0],[9E9,9E9,9E9,9E9,9E9,9E9]];
            P05W07_ArcEnd := [[0,0,0],[1,0,0,0],[0,0,0,0],[9E9,9E9,9E9,9E9,9E9,9E9]];
            P05W07_Approach := [[0,0,0],[1,0,0,0],[0,0,0,0],[9E9,9E9,9E9,9E9,9E9,9E9]];
            P05W07_Retract := [[0,0,0],[1,0,0,0],[0,0,0,0],[9E9,9E9,9E9,9E9,9E9,9E9]];
            P05W07_Trans := [[0,0,0],[1,0,0,0],[0,0,0,0],[9E9,9E9,9E9,9E9,9E9,9E9]];
        ELSEIF slot = 8 THEN
            P05W08_Used := FALSE;
            P05W08_SubType := 0;
            P05W08_ToolSel := 0;
            P05W08_LenMM := 0;
            P05W08_ArcStart := [[0,0,0],[1,0,0,0],[0,0,0,0],[9E9,9E9,9E9,9E9,9E9,9E9]];
            P05W08_ArcEnd := [[0,0,0],[1,0,0,0],[0,0,0,0],[9E9,9E9,9E9,9E9,9E9,9E9]];
            P05W08_Approach := [[0,0,0],[1,0,0,0],[0,0,0,0],[9E9,9E9,9E9,9E9,9E9,9E9]];
            P05W08_Retract := [[0,0,0],[1,0,0,0],[0,0,0,0],[9E9,9E9,9E9,9E9,9E9,9E9]];
            P05W08_Trans := [[0,0,0],[1,0,0,0],[0,0,0,0],[9E9,9E9,9E9,9E9,9E9,9E9]];
        ELSEIF slot = 9 THEN
            P05W09_Used := FALSE;
            P05W09_SubType := 0;
            P05W09_ToolSel := 0;
            P05W09_LenMM := 0;
            P05W09_ArcStart := [[0,0,0],[1,0,0,0],[0,0,0,0],[9E9,9E9,9E9,9E9,9E9,9E9]];
            P05W09_ArcEnd := [[0,0,0],[1,0,0,0],[0,0,0,0],[9E9,9E9,9E9,9E9,9E9,9E9]];
            P05W09_Approach := [[0,0,0],[1,0,0,0],[0,0,0,0],[9E9,9E9,9E9,9E9,9E9,9E9]];
            P05W09_Retract := [[0,0,0],[1,0,0,0],[0,0,0,0],[9E9,9E9,9E9,9E9,9E9,9E9]];
            P05W09_Trans := [[0,0,0],[1,0,0,0],[0,0,0,0],[9E9,9E9,9E9,9E9,9E9,9E9]];
        ELSEIF slot = 10 THEN
            P05W10_Used := FALSE;
            P05W10_SubType := 0;
            P05W10_ToolSel := 0;
            P05W10_LenMM := 0;
            P05W10_ArcStart := [[0,0,0],[1,0,0,0],[0,0,0,0],[9E9,9E9,9E9,9E9,9E9,9E9]];
            P05W10_ArcEnd := [[0,0,0],[1,0,0,0],[0,0,0,0],[9E9,9E9,9E9,9E9,9E9,9E9]];
            P05W10_Approach := [[0,0,0],[1,0,0,0],[0,0,0,0],[9E9,9E9,9E9,9E9,9E9,9E9]];
            P05W10_Retract := [[0,0,0],[1,0,0,0],[0,0,0,0],[9E9,9E9,9E9,9E9,9E9,9E9]];
            P05W10_Trans := [[0,0,0],[1,0,0,0],[0,0,0,0],[9E9,9E9,9E9,9E9,9E9,9E9]];
        ELSEIF slot = 11 THEN
            P05W11_Used := FALSE;
            P05W11_SubType := 0;
            P05W11_ToolSel := 0;
            P05W11_LenMM := 0;
            P05W11_ArcStart := [[0,0,0],[1,0,0,0],[0,0,0,0],[9E9,9E9,9E9,9E9,9E9,9E9]];
            P05W11_ArcEnd := [[0,0,0],[1,0,0,0],[0,0,0,0],[9E9,9E9,9E9,9E9,9E9,9E9]];
            P05W11_Approach := [[0,0,0],[1,0,0,0],[0,0,0,0],[9E9,9E9,9E9,9E9,9E9,9E9]];
            P05W11_Retract := [[0,0,0],[1,0,0,0],[0,0,0,0],[9E9,9E9,9E9,9E9,9E9,9E9]];
            P05W11_Trans := [[0,0,0],[1,0,0,0],[0,0,0,0],[9E9,9E9,9E9,9E9,9E9,9E9]];
        ELSEIF slot = 12 THEN
            P05W12_Used := FALSE;
            P05W12_SubType := 0;
            P05W12_ToolSel := 0;
            P05W12_LenMM := 0;
            P05W12_ArcStart := [[0,0,0],[1,0,0,0],[0,0,0,0],[9E9,9E9,9E9,9E9,9E9,9E9]];
            P05W12_ArcEnd := [[0,0,0],[1,0,0,0],[0,0,0,0],[9E9,9E9,9E9,9E9,9E9,9E9]];
            P05W12_Approach := [[0,0,0],[1,0,0,0],[0,0,0,0],[9E9,9E9,9E9,9E9,9E9,9E9]];
            P05W12_Retract := [[0,0,0],[1,0,0,0],[0,0,0,0],[9E9,9E9,9E9,9E9,9E9,9E9]];
            P05W12_Trans := [[0,0,0],[1,0,0,0],[0,0,0,0],[9E9,9E9,9E9,9E9,9E9,9E9]];
        ELSEIF slot = 13 THEN
            P05W13_Used := FALSE;
            P05W13_SubType := 0;
            P05W13_ToolSel := 0;
            P05W13_LenMM := 0;
            P05W13_ArcStart := [[0,0,0],[1,0,0,0],[0,0,0,0],[9E9,9E9,9E9,9E9,9E9,9E9]];
            P05W13_ArcEnd := [[0,0,0],[1,0,0,0],[0,0,0,0],[9E9,9E9,9E9,9E9,9E9,9E9]];
            P05W13_Approach := [[0,0,0],[1,0,0,0],[0,0,0,0],[9E9,9E9,9E9,9E9,9E9,9E9]];
            P05W13_Retract := [[0,0,0],[1,0,0,0],[0,0,0,0],[9E9,9E9,9E9,9E9,9E9,9E9]];
            P05W13_Trans := [[0,0,0],[1,0,0,0],[0,0,0,0],[9E9,9E9,9E9,9E9,9E9,9E9]];
        ELSEIF slot = 14 THEN
            P05W14_Used := FALSE;
            P05W14_SubType := 0;
            P05W14_ToolSel := 0;
            P05W14_LenMM := 0;
            P05W14_ArcStart := [[0,0,0],[1,0,0,0],[0,0,0,0],[9E9,9E9,9E9,9E9,9E9,9E9]];
            P05W14_ArcEnd := [[0,0,0],[1,0,0,0],[0,0,0,0],[9E9,9E9,9E9,9E9,9E9,9E9]];
            P05W14_Approach := [[0,0,0],[1,0,0,0],[0,0,0,0],[9E9,9E9,9E9,9E9,9E9,9E9]];
            P05W14_Retract := [[0,0,0],[1,0,0,0],[0,0,0,0],[9E9,9E9,9E9,9E9,9E9,9E9]];
            P05W14_Trans := [[0,0,0],[1,0,0,0],[0,0,0,0],[9E9,9E9,9E9,9E9,9E9,9E9]];
        ELSEIF slot = 15 THEN
            P05W15_Used := FALSE;
            P05W15_SubType := 0;
            P05W15_ToolSel := 0;
            P05W15_LenMM := 0;
            P05W15_ArcStart := [[0,0,0],[1,0,0,0],[0,0,0,0],[9E9,9E9,9E9,9E9,9E9,9E9]];
            P05W15_ArcEnd := [[0,0,0],[1,0,0,0],[0,0,0,0],[9E9,9E9,9E9,9E9,9E9,9E9]];
            P05W15_Approach := [[0,0,0],[1,0,0,0],[0,0,0,0],[9E9,9E9,9E9,9E9,9E9,9E9]];
            P05W15_Retract := [[0,0,0],[1,0,0,0],[0,0,0,0],[9E9,9E9,9E9,9E9,9E9,9E9]];
            P05W15_Trans := [[0,0,0],[1,0,0,0],[0,0,0,0],[9E9,9E9,9E9,9E9,9E9,9E9]];
        ELSEIF slot = 16 THEN
            P05W16_Used := FALSE;
            P05W16_SubType := 0;
            P05W16_ToolSel := 0;
            P05W16_LenMM := 0;
            P05W16_ArcStart := [[0,0,0],[1,0,0,0],[0,0,0,0],[9E9,9E9,9E9,9E9,9E9,9E9]];
            P05W16_ArcEnd := [[0,0,0],[1,0,0,0],[0,0,0,0],[9E9,9E9,9E9,9E9,9E9,9E9]];
            P05W16_Approach := [[0,0,0],[1,0,0,0],[0,0,0,0],[9E9,9E9,9E9,9E9,9E9,9E9]];
            P05W16_Retract := [[0,0,0],[1,0,0,0],[0,0,0,0],[9E9,9E9,9E9,9E9,9E9,9E9]];
            P05W16_Trans := [[0,0,0],[1,0,0,0],[0,0,0,0],[9E9,9E9,9E9,9E9,9E9,9E9]];
        ELSEIF slot = 17 THEN
            P05W17_Used := FALSE;
            P05W17_SubType := 0;
            P05W17_ToolSel := 0;
            P05W17_LenMM := 0;
            P05W17_ArcStart := [[0,0,0],[1,0,0,0],[0,0,0,0],[9E9,9E9,9E9,9E9,9E9,9E9]];
            P05W17_ArcEnd := [[0,0,0],[1,0,0,0],[0,0,0,0],[9E9,9E9,9E9,9E9,9E9,9E9]];
            P05W17_Approach := [[0,0,0],[1,0,0,0],[0,0,0,0],[9E9,9E9,9E9,9E9,9E9,9E9]];
            P05W17_Retract := [[0,0,0],[1,0,0,0],[0,0,0,0],[9E9,9E9,9E9,9E9,9E9,9E9]];
            P05W17_Trans := [[0,0,0],[1,0,0,0],[0,0,0,0],[9E9,9E9,9E9,9E9,9E9,9E9]];
        ELSEIF slot = 18 THEN
            P05W18_Used := FALSE;
            P05W18_SubType := 0;
            P05W18_ToolSel := 0;
            P05W18_LenMM := 0;
            P05W18_ArcStart := [[0,0,0],[1,0,0,0],[0,0,0,0],[9E9,9E9,9E9,9E9,9E9,9E9]];
            P05W18_ArcEnd := [[0,0,0],[1,0,0,0],[0,0,0,0],[9E9,9E9,9E9,9E9,9E9,9E9]];
            P05W18_Approach := [[0,0,0],[1,0,0,0],[0,0,0,0],[9E9,9E9,9E9,9E9,9E9,9E9]];
            P05W18_Retract := [[0,0,0],[1,0,0,0],[0,0,0,0],[9E9,9E9,9E9,9E9,9E9,9E9]];
            P05W18_Trans := [[0,0,0],[1,0,0,0],[0,0,0,0],[9E9,9E9,9E9,9E9,9E9,9E9]];
        ELSEIF slot = 19 THEN
            P05W19_Used := FALSE;
            P05W19_SubType := 0;
            P05W19_ToolSel := 0;
            P05W19_LenMM := 0;
            P05W19_ArcStart := [[0,0,0],[1,0,0,0],[0,0,0,0],[9E9,9E9,9E9,9E9,9E9,9E9]];
            P05W19_ArcEnd := [[0,0,0],[1,0,0,0],[0,0,0,0],[9E9,9E9,9E9,9E9,9E9,9E9]];
            P05W19_Approach := [[0,0,0],[1,0,0,0],[0,0,0,0],[9E9,9E9,9E9,9E9,9E9,9E9]];
            P05W19_Retract := [[0,0,0],[1,0,0,0],[0,0,0,0],[9E9,9E9,9E9,9E9,9E9,9E9]];
            P05W19_Trans := [[0,0,0],[1,0,0,0],[0,0,0,0],[9E9,9E9,9E9,9E9,9E9,9E9]];
        ELSEIF slot = 20 THEN
            P05W20_Used := FALSE;
            P05W20_SubType := 0;
            P05W20_ToolSel := 0;
            P05W20_LenMM := 0;
            P05W20_ArcStart := [[0,0,0],[1,0,0,0],[0,0,0,0],[9E9,9E9,9E9,9E9,9E9,9E9]];
            P05W20_ArcEnd := [[0,0,0],[1,0,0,0],[0,0,0,0],[9E9,9E9,9E9,9E9,9E9,9E9]];
            P05W20_Approach := [[0,0,0],[1,0,0,0],[0,0,0,0],[9E9,9E9,9E9,9E9,9E9,9E9]];
            P05W20_Retract := [[0,0,0],[1,0,0,0],[0,0,0,0],[9E9,9E9,9E9,9E9,9E9,9E9]];
            P05W20_Trans := [[0,0,0],[1,0,0,0],[0,0,0,0],[9E9,9E9,9E9,9E9,9E9,9E9]];
        ELSEIF slot = 21 THEN
            P05W21_Used := FALSE;
            P05W21_SubType := 0;
            P05W21_ToolSel := 0;
            P05W21_LenMM := 0;
            P05W21_ArcStart := [[0,0,0],[1,0,0,0],[0,0,0,0],[9E9,9E9,9E9,9E9,9E9,9E9]];
            P05W21_ArcEnd := [[0,0,0],[1,0,0,0],[0,0,0,0],[9E9,9E9,9E9,9E9,9E9,9E9]];
            P05W21_Approach := [[0,0,0],[1,0,0,0],[0,0,0,0],[9E9,9E9,9E9,9E9,9E9,9E9]];
            P05W21_Retract := [[0,0,0],[1,0,0,0],[0,0,0,0],[9E9,9E9,9E9,9E9,9E9,9E9]];
            P05W21_Trans := [[0,0,0],[1,0,0,0],[0,0,0,0],[9E9,9E9,9E9,9E9,9E9,9E9]];
        ELSEIF slot = 22 THEN
            P05W22_Used := FALSE;
            P05W22_SubType := 0;
            P05W22_ToolSel := 0;
            P05W22_LenMM := 0;
            P05W22_ArcStart := [[0,0,0],[1,0,0,0],[0,0,0,0],[9E9,9E9,9E9,9E9,9E9,9E9]];
            P05W22_ArcEnd := [[0,0,0],[1,0,0,0],[0,0,0,0],[9E9,9E9,9E9,9E9,9E9,9E9]];
            P05W22_Approach := [[0,0,0],[1,0,0,0],[0,0,0,0],[9E9,9E9,9E9,9E9,9E9,9E9]];
            P05W22_Retract := [[0,0,0],[1,0,0,0],[0,0,0,0],[9E9,9E9,9E9,9E9,9E9,9E9]];
            P05W22_Trans := [[0,0,0],[1,0,0,0],[0,0,0,0],[9E9,9E9,9E9,9E9,9E9,9E9]];
        ELSEIF slot = 23 THEN
            P05W23_Used := FALSE;
            P05W23_SubType := 0;
            P05W23_ToolSel := 0;
            P05W23_LenMM := 0;
            P05W23_ArcStart := [[0,0,0],[1,0,0,0],[0,0,0,0],[9E9,9E9,9E9,9E9,9E9,9E9]];
            P05W23_ArcEnd := [[0,0,0],[1,0,0,0],[0,0,0,0],[9E9,9E9,9E9,9E9,9E9,9E9]];
            P05W23_Approach := [[0,0,0],[1,0,0,0],[0,0,0,0],[9E9,9E9,9E9,9E9,9E9,9E9]];
            P05W23_Retract := [[0,0,0],[1,0,0,0],[0,0,0,0],[9E9,9E9,9E9,9E9,9E9,9E9]];
            P05W23_Trans := [[0,0,0],[1,0,0,0],[0,0,0,0],[9E9,9E9,9E9,9E9,9E9,9E9]];
        ELSEIF slot = 24 THEN
            P05W24_Used := FALSE;
            P05W24_SubType := 0;
            P05W24_ToolSel := 0;
            P05W24_LenMM := 0;
            P05W24_ArcStart := [[0,0,0],[1,0,0,0],[0,0,0,0],[9E9,9E9,9E9,9E9,9E9,9E9]];
            P05W24_ArcEnd := [[0,0,0],[1,0,0,0],[0,0,0,0],[9E9,9E9,9E9,9E9,9E9,9E9]];
            P05W24_Approach := [[0,0,0],[1,0,0,0],[0,0,0,0],[9E9,9E9,9E9,9E9,9E9,9E9]];
            P05W24_Retract := [[0,0,0],[1,0,0,0],[0,0,0,0],[9E9,9E9,9E9,9E9,9E9,9E9]];
            P05W24_Trans := [[0,0,0],[1,0,0,0],[0,0,0,0],[9E9,9E9,9E9,9E9,9E9,9E9]];
        ELSEIF slot = 25 THEN
            P05W25_Used := FALSE;
            P05W25_SubType := 0;
            P05W25_ToolSel := 0;
            P05W25_LenMM := 0;
            P05W25_ArcStart := [[0,0,0],[1,0,0,0],[0,0,0,0],[9E9,9E9,9E9,9E9,9E9,9E9]];
            P05W25_ArcEnd := [[0,0,0],[1,0,0,0],[0,0,0,0],[9E9,9E9,9E9,9E9,9E9,9E9]];
            P05W25_Approach := [[0,0,0],[1,0,0,0],[0,0,0,0],[9E9,9E9,9E9,9E9,9E9,9E9]];
            P05W25_Retract := [[0,0,0],[1,0,0,0],[0,0,0,0],[9E9,9E9,9E9,9E9,9E9,9E9]];
            P05W25_Trans := [[0,0,0],[1,0,0,0],[0,0,0,0],[9E9,9E9,9E9,9E9,9E9,9E9]];
        ELSEIF slot = 26 THEN
            P05W26_Used := FALSE;
            P05W26_SubType := 0;
            P05W26_ToolSel := 0;
            P05W26_LenMM := 0;
            P05W26_ArcStart := [[0,0,0],[1,0,0,0],[0,0,0,0],[9E9,9E9,9E9,9E9,9E9,9E9]];
            P05W26_ArcEnd := [[0,0,0],[1,0,0,0],[0,0,0,0],[9E9,9E9,9E9,9E9,9E9,9E9]];
            P05W26_Approach := [[0,0,0],[1,0,0,0],[0,0,0,0],[9E9,9E9,9E9,9E9,9E9,9E9]];
            P05W26_Retract := [[0,0,0],[1,0,0,0],[0,0,0,0],[9E9,9E9,9E9,9E9,9E9,9E9]];
            P05W26_Trans := [[0,0,0],[1,0,0,0],[0,0,0,0],[9E9,9E9,9E9,9E9,9E9,9E9]];
        ELSEIF slot = 27 THEN
            P05W27_Used := FALSE;
            P05W27_SubType := 0;
            P05W27_ToolSel := 0;
            P05W27_LenMM := 0;
            P05W27_ArcStart := [[0,0,0],[1,0,0,0],[0,0,0,0],[9E9,9E9,9E9,9E9,9E9,9E9]];
            P05W27_ArcEnd := [[0,0,0],[1,0,0,0],[0,0,0,0],[9E9,9E9,9E9,9E9,9E9,9E9]];
            P05W27_Approach := [[0,0,0],[1,0,0,0],[0,0,0,0],[9E9,9E9,9E9,9E9,9E9,9E9]];
            P05W27_Retract := [[0,0,0],[1,0,0,0],[0,0,0,0],[9E9,9E9,9E9,9E9,9E9,9E9]];
            P05W27_Trans := [[0,0,0],[1,0,0,0],[0,0,0,0],[9E9,9E9,9E9,9E9,9E9,9E9]];
        ELSEIF slot = 28 THEN
            P05W28_Used := FALSE;
            P05W28_SubType := 0;
            P05W28_ToolSel := 0;
            P05W28_LenMM := 0;
            P05W28_ArcStart := [[0,0,0],[1,0,0,0],[0,0,0,0],[9E9,9E9,9E9,9E9,9E9,9E9]];
            P05W28_ArcEnd := [[0,0,0],[1,0,0,0],[0,0,0,0],[9E9,9E9,9E9,9E9,9E9,9E9]];
            P05W28_Approach := [[0,0,0],[1,0,0,0],[0,0,0,0],[9E9,9E9,9E9,9E9,9E9,9E9]];
            P05W28_Retract := [[0,0,0],[1,0,0,0],[0,0,0,0],[9E9,9E9,9E9,9E9,9E9,9E9]];
            P05W28_Trans := [[0,0,0],[1,0,0,0],[0,0,0,0],[9E9,9E9,9E9,9E9,9E9,9E9]];
        ELSEIF slot = 29 THEN
            P05W29_Used := FALSE;
            P05W29_SubType := 0;
            P05W29_ToolSel := 0;
            P05W29_LenMM := 0;
            P05W29_ArcStart := [[0,0,0],[1,0,0,0],[0,0,0,0],[9E9,9E9,9E9,9E9,9E9,9E9]];
            P05W29_ArcEnd := [[0,0,0],[1,0,0,0],[0,0,0,0],[9E9,9E9,9E9,9E9,9E9,9E9]];
            P05W29_Approach := [[0,0,0],[1,0,0,0],[0,0,0,0],[9E9,9E9,9E9,9E9,9E9,9E9]];
            P05W29_Retract := [[0,0,0],[1,0,0,0],[0,0,0,0],[9E9,9E9,9E9,9E9,9E9,9E9]];
            P05W29_Trans := [[0,0,0],[1,0,0,0],[0,0,0,0],[9E9,9E9,9E9,9E9,9E9,9E9]];
        ELSEIF slot = 30 THEN
            P05W30_Used := FALSE;
            P05W30_SubType := 0;
            P05W30_ToolSel := 0;
            P05W30_LenMM := 0;
            P05W30_ArcStart := [[0,0,0],[1,0,0,0],[0,0,0,0],[9E9,9E9,9E9,9E9,9E9,9E9]];
            P05W30_ArcEnd := [[0,0,0],[1,0,0,0],[0,0,0,0],[9E9,9E9,9E9,9E9,9E9,9E9]];
            P05W30_Approach := [[0,0,0],[1,0,0,0],[0,0,0,0],[9E9,9E9,9E9,9E9,9E9,9E9]];
            P05W30_Retract := [[0,0,0],[1,0,0,0],[0,0,0,0],[9E9,9E9,9E9,9E9,9E9,9E9]];
            P05W30_Trans := [[0,0,0],[1,0,0,0],[0,0,0,0],[9E9,9E9,9E9,9E9,9E9,9E9]];
        ELSE
            TPWrite "Invalid weld slot.";
        ENDIF
    ENDPROC

    PROC StoreNextFree_P05(num subType, num toolSel, num lenMM,
                       robtarget arcStart, robtarget arcEnd, robtarget approach, robtarget retract, robtarget trans)
        IF NOT P05W01_Used THEN
            StoreSlot_P05 1, subType, toolSel, lenMM, arcStart, arcEnd, approach, retract, trans;
            nWeldsP05 := nWeldsP05 + 1;
            RETURN;
        ELSEIF NOT P05W02_Used THEN
            StoreSlot_P05 2, subType, toolSel, lenMM, arcStart, arcEnd, approach, retract, trans;
            nWeldsP05 := nWeldsP05 + 1;
            RETURN;
        ELSEIF NOT P05W03_Used THEN
            StoreSlot_P05 3, subType, toolSel, lenMM, arcStart, arcEnd, approach, retract, trans;
            nWeldsP05 := nWeldsP05 + 1;
            RETURN;
        ELSEIF NOT P05W04_Used THEN
            StoreSlot_P05 4, subType, toolSel, lenMM, arcStart, arcEnd, approach, retract, trans;
            nWeldsP05 := nWeldsP05 + 1;
            RETURN;
        ELSEIF NOT P05W05_Used THEN
            StoreSlot_P05 5, subType, toolSel, lenMM, arcStart, arcEnd, approach, retract, trans;
            nWeldsP05 := nWeldsP05 + 1;
            RETURN;
        ELSEIF NOT P05W06_Used THEN
            StoreSlot_P05 6, subType, toolSel, lenMM, arcStart, arcEnd, approach, retract, trans;
            nWeldsP05 := nWeldsP05 + 1;
            RETURN;
        ELSEIF NOT P05W07_Used THEN
            StoreSlot_P05 7, subType, toolSel, lenMM, arcStart, arcEnd, approach, retract, trans;
            nWeldsP05 := nWeldsP05 + 1;
            RETURN;
        ELSEIF NOT P05W08_Used THEN
            StoreSlot_P05 8, subType, toolSel, lenMM, arcStart, arcEnd, approach, retract, trans;
            nWeldsP05 := nWeldsP05 + 1;
            RETURN;
        ELSEIF NOT P05W09_Used THEN
            StoreSlot_P05 9, subType, toolSel, lenMM, arcStart, arcEnd, approach, retract, trans;
            nWeldsP05 := nWeldsP05 + 1;
            RETURN;
        ELSEIF NOT P05W10_Used THEN
            StoreSlot_P05 10, subType, toolSel, lenMM, arcStart, arcEnd, approach, retract, trans;
            nWeldsP05 := nWeldsP05 + 1;
            RETURN;
        ELSEIF NOT P05W11_Used THEN
            StoreSlot_P05 11, subType, toolSel, lenMM, arcStart, arcEnd, approach, retract, trans;
            nWeldsP05 := nWeldsP05 + 1;
            RETURN;
        ELSEIF NOT P05W12_Used THEN
            StoreSlot_P05 12, subType, toolSel, lenMM, arcStart, arcEnd, approach, retract, trans;
            nWeldsP05 := nWeldsP05 + 1;
            RETURN;
        ELSEIF NOT P05W13_Used THEN
            StoreSlot_P05 13, subType, toolSel, lenMM, arcStart, arcEnd, approach, retract, trans;
            nWeldsP05 := nWeldsP05 + 1;
            RETURN;
        ELSEIF NOT P05W14_Used THEN
            StoreSlot_P05 14, subType, toolSel, lenMM, arcStart, arcEnd, approach, retract, trans;
            nWeldsP05 := nWeldsP05 + 1;
            RETURN;
        ELSEIF NOT P05W15_Used THEN
            StoreSlot_P05 15, subType, toolSel, lenMM, arcStart, arcEnd, approach, retract, trans;
            nWeldsP05 := nWeldsP05 + 1;
            RETURN;
        ELSEIF NOT P05W16_Used THEN
            StoreSlot_P05 16, subType, toolSel, lenMM, arcStart, arcEnd, approach, retract, trans;
            nWeldsP05 := nWeldsP05 + 1;
            RETURN;
        ELSEIF NOT P05W17_Used THEN
            StoreSlot_P05 17, subType, toolSel, lenMM, arcStart, arcEnd, approach, retract, trans;
            nWeldsP05 := nWeldsP05 + 1;
            RETURN;
        ELSEIF NOT P05W18_Used THEN
            StoreSlot_P05 18, subType, toolSel, lenMM, arcStart, arcEnd, approach, retract, trans;
            nWeldsP05 := nWeldsP05 + 1;
            RETURN;
        ELSEIF NOT P05W19_Used THEN
            StoreSlot_P05 19, subType, toolSel, lenMM, arcStart, arcEnd, approach, retract, trans;
            nWeldsP05 := nWeldsP05 + 1;
            RETURN;
        ELSEIF NOT P05W20_Used THEN
            StoreSlot_P05 20, subType, toolSel, lenMM, arcStart, arcEnd, approach, retract, trans;
            nWeldsP05 := nWeldsP05 + 1;
            RETURN;
        ELSEIF NOT P05W21_Used THEN
            StoreSlot_P05 21, subType, toolSel, lenMM, arcStart, arcEnd, approach, retract, trans;
            nWeldsP05 := nWeldsP05 + 1;
            RETURN;
        ELSEIF NOT P05W22_Used THEN
            StoreSlot_P05 22, subType, toolSel, lenMM, arcStart, arcEnd, approach, retract, trans;
            nWeldsP05 := nWeldsP05 + 1;
            RETURN;
        ELSEIF NOT P05W23_Used THEN
            StoreSlot_P05 23, subType, toolSel, lenMM, arcStart, arcEnd, approach, retract, trans;
            nWeldsP05 := nWeldsP05 + 1;
            RETURN;
        ELSEIF NOT P05W24_Used THEN
            StoreSlot_P05 24, subType, toolSel, lenMM, arcStart, arcEnd, approach, retract, trans;
            nWeldsP05 := nWeldsP05 + 1;
            RETURN;
        ELSEIF NOT P05W25_Used THEN
            StoreSlot_P05 25, subType, toolSel, lenMM, arcStart, arcEnd, approach, retract, trans;
            nWeldsP05 := nWeldsP05 + 1;
            RETURN;
        ELSEIF NOT P05W26_Used THEN
            StoreSlot_P05 26, subType, toolSel, lenMM, arcStart, arcEnd, approach, retract, trans;
            nWeldsP05 := nWeldsP05 + 1;
            RETURN;
        ELSEIF NOT P05W27_Used THEN
            StoreSlot_P05 27, subType, toolSel, lenMM, arcStart, arcEnd, approach, retract, trans;
            nWeldsP05 := nWeldsP05 + 1;
            RETURN;
        ELSEIF NOT P05W28_Used THEN
            StoreSlot_P05 28, subType, toolSel, lenMM, arcStart, arcEnd, approach, retract, trans;
            nWeldsP05 := nWeldsP05 + 1;
            RETURN;
        ELSEIF NOT P05W29_Used THEN
            StoreSlot_P05 29, subType, toolSel, lenMM, arcStart, arcEnd, approach, retract, trans;
            nWeldsP05 := nWeldsP05 + 1;
            RETURN;
        ELSEIF NOT P05W30_Used THEN
            StoreSlot_P05 30, subType, toolSel, lenMM, arcStart, arcEnd, approach, retract, trans;
            nWeldsP05 := nWeldsP05 + 1;
            RETURN;
        ELSE
            TPWrite "No free weld slots available.";
        ENDIF
    ENDPROC

